// TIA Portal project "1905391_000_019" (V16)

(* hardware
DEVICE "S7-1200 station_1"  S7-1200 Station
   slot 0: "Rack_0"  S7-1200 Rack  Rack  V1.0
   slot 1: "PLC_1"  CPU 1211C DC/DC/DC  6ES7 211-1AE40-0XB0  V4.4
DEVICE "HMI_1"  TP900 Comfort
   slot 0: "HMI_1"  TP900 Comfort  6AV2 124-0JC01-0AX0  16.0.0.0
   slot 1: "HMI_RT_1"  TP900 Comfort  6AV2 124-0JC01-0AX0  16.0.0.0
   slot 5: "HMI_1.IE_CP_1"  PROFINET Interface  16.0.0.0
      slot 1: "PROFINET Interface_1"  PROFINET Interface
         slot 1: "Port_1"  Port
         slot 2: "Port_2"  Port
   slot 7: "HMI_1.MPI/DP_CP_1"  MPI/DP Interface  16.0.0.0
*)

// ===== PLC "PLC_1"  CPU 1211C DC/DC/DC =====

VAR_GLOBAL   // PLC tag table "Default tag table"
   "System_Byte" AT %MB1 : Byte;
   "FirstScan" AT %M1.0 : Bool;
   "DiagStatusUpdate" AT %M1.1 : Bool;
   "AlwaysTRUE" AT %M1.2 : Bool;
   "AlwaysFALSE" AT %M1.3 : Bool;
   "Clock_Byte" AT %MB0 : Byte;
   "Clock_10Hz" AT %M0.0 : Bool;
   "Clock_5Hz" AT %M0.1 : Bool;
   "Clock_2.5Hz" AT %M0.2 : Bool;
   "Clock_2Hz" AT %M0.3 : Bool;
   "Clock_1.25Hz" AT %M0.4 : Bool;
   "Clock_1Hz" AT %M0.5 : Bool;
   "Clock_0.625Hz" AT %M0.6 : Bool;
   "Clock_0.5Hz" AT %M0.7 : Bool;
END_VAR

VAR_GLOBAL CONSTANT   // PLC tag table "Default tag table"
   "STRING_LENGTH" : Int := 20;
   "ADP_PARAMETER_LENGTH" : Int := 5;
   "NULL_TOKEN" : Int := -1;
END_VAR

VAR_GLOBAL CONSTANT   // PLC tag table "Colors"
   "LABEL_COLOR" : String := '200_200_200';
   "DESELECTED_INPUT_COOR" : String := '250_250_250';
   "SELECTED_INPUT_COLOR" : String := '150,250,150';
   "BORDER_COLOR" : String := '200_200_200';
   "DIVIDER_COLOR" : String := '50_75_100';
   "THIS_SCREEN_COLOR" : String := '150;150;150';
   "OTHER_SCREEN_COLOR" : String := '100,100,100';
   "NAVIGATION_ACTUATE" : String := '150_250_150';
   "BACKGROUND_COLOR" : String := '150,150,200';
END_VAR

VAR_GLOBAL CONSTANT   // PLC tag table "Screen_Numbers"
   "WIRES_SCREEN_NUMBER" : Int := 1;
   "MATERIALS_SCREEN_NUMBER" : Int := 2;
END_VAR

TYPE "Divider.UDT"
   STRUCT
      background_animate : DInt;
      background_visible : Bool;
      line_animate : DInt;
      line_visible : Bool;
   END_STRUCT;
END_TYPE

TYPE "Row_Data.UDT"
   STRUCT
      background_animate : DInt;
      background_visible : Bool;
      cell_0_animate : DInt;
      cell_0_visible : Bool;
      cell_1_active : Bool;
      cell_1_animate : DInt;
      cell_1_enable : Bool;
      cell_1_input_finished : Bool;
      cell_1_value : String[50];
      cell_1_visible : Bool;
   END_STRUCT;
END_TYPE

TYPE "HMI_Interface.UDT"
   STRUCT
      materials : "Materials.HMI.UDT";
      meta : "HMI_Meta.UDT";
      navigation : "Navigation.HMI.UDT";
      wires : "Wire.HMI.UDT";
   END_STRUCT;
END_TYPE

TYPE "LED_Interface.UDT"
   STRUCT
      elements : "Material.LED.UDT";
      wires : "Wires.LED.UDT";
   END_STRUCT;
END_TYPE

TYPE "Navigation.HMI.UDT"
   STRUCT
      background_animate : DInt;
      background_visible : Bool;
      bottom_line_animate : DInt;
      bottom_line_visible : Bool;
      material_actuate : Bool;
      material_animate : DInt;
      material_cover_animate : DInt;
      material_cover_visible : Bool;
      material_enable : Bool;
      material_visible : Bool;
      wire_actuate : Bool;
      wire_animate : DInt;
      wire_cover_animate : DInt;
      wire_cover_visible : Bool;
      wire_enable : Bool;
      wire_visible : Bool;
   END_STRUCT;
END_TYPE

TYPE "Row_Custom.UDT"
   STRUCT
      background_animate : DInt;
      background_visible : Bool;
      cell_0_activate : Bool;
      cell_0_animate : DInt;
      cell_0_enable : Bool;
      cell_0_input_finished : Bool;
      cell_0_value : String[50];
      cell_0_visible : Bool;
      cell_1_activate : Bool;
      cell_1_animate : DInt;
      cell_1_enable : Bool;
      cell_1_input_finished : Bool;
      cell_1_value : String[50];
      cell_1_visible : Bool;
   END_STRUCT;
END_TYPE

TYPE "Row_Label.UDT"
   STRUCT
      background_animate : DInt;
      background_visible : Bool;
      cell_0_animate : DInt;
      cell_0_visible : Bool;
      cell_1_animate : DInt;
      cell_1_visible : Bool;
   END_STRUCT;
END_TYPE

TYPE "HMI_Meta.UDT"
   STRUCT
      screen_number : Int;
   END_STRUCT;
END_TYPE

TYPE "Screen_Background.UDT"
   STRUCT
      color : DInt;
      visible : Bool;
   END_STRUCT;
END_TYPE

// folder: ADP Data

TYPE "ADP.Row.2_Cells.UDT"
   STRUCT
      me : Array[0..1] of "ADP.Cell.UDT";
   END_STRUCT;
END_TYPE

TYPE "ADP.Cell.UDT"
   STRUCT
      color : String["ADP_PARAMETER_LENGTH"];
      flashing : String["ADP_PARAMETER_LENGTH"];
      h_align : String["ADP_PARAMETER_LENGTH"];
      lince_control : String["ADP_PARAMETER_LENGTH"];
      scroll_speed : String["ADP_PARAMETER_LENGTH"];
      size_and_face : String["ADP_PARAMETER_LENGTH"];
      v_align : String["ADP_PARAMETER_LENGTH"];
      value : String["STRING_LENGTH"];
   END_STRUCT;
END_TYPE

TYPE "ADP.Message_Buffer.UDT"
   STRUCT
      me : Array[0..999] of Byte;
   END_STRUCT;
END_TYPE

TYPE "ADP.Decoded.UDT"
   STRUCT
      color : "ADP.Decoded.Color.UDT";
      flash : "ADP.Decoded.Flash.UDT";
      horizontal_alignment : "ADP.Decoded.Horizontal_Alignment.UDT";
      line_control : "ADP.Decoded.Line_Control.UDT";
      scroll_speed : "ADP.Decoded.Scroll_Speed.UDT";
      size_and_face : "ADP.Decoded.Size_and_Face.UDT";
      vertical_alignment : "ADP.Decoded.Vertical_Alignment.UDT";
   END_STRUCT;
END_TYPE

TYPE "ADP.Decoded.Color.UDT"
   STRUCT
      black : String[8] := 'black';
      blue : String[8] := 'blue';
      green : String[8] := 'green';
      mix_1 : String[8] := 'mix 1';
      mix_2 : String[8] := 'mix 2';
      mix_3 : String[8] := 'mix 3';
      mix_4 : String[8] := 'mix 4';
      red : String[8] := 'red';
      white : String[8] := 'white';
      yellow : String[8] := 'yellow';
   END_STRUCT;
END_TYPE

TYPE "ADP.Decoded.Flash.UDT"
   STRUCT
      off : String[8] := 'off';
      on : String[8] := 'on';
   END_STRUCT;
END_TYPE

TYPE "ADP.Decoded.Horizontal_Alignment.UDT"
   STRUCT
      center : String[8] := 'center';
      left : String[8] := 'left';
      right : String[8] := 'right';
   END_STRUCT;
END_TYPE

TYPE "ADP.Encoded.UDT"
VERSION : 0.1
   STRUCT
      file_system : "ADP.Encoded.File_System.UDT";
      formatting : "ADP.Encoded.Formatting.UDT";
   END_STRUCT;
END_TYPE

TYPE "ADP.Message_Formats.Encoded.UDT"
   STRUCT
      color : String [5];
      flash : String [5];
      scroll_speed : String [5];
      size_and_face : String [5];
      vertical_alignment : String [5];
      horizontal_alignment : String [5];
   END_STRUCT;
END_TYPE

TYPE "ADP.Message_Formats.Decoded.UDT"
   STRUCT
      color : String [20];
      flash : String [20];
      scroll_speed : String [20];
      size_and_face : String [20];
      vertical_alignment : String [20];
      horizontal_alignment : String [20];
   END_STRUCT;
END_TYPE

TYPE "ADP.Decoded.Scroll_Speed.UDT"
   STRUCT
      slowest : String[9] := 'slowest';
      slow : String[9] := 'slow';
      normal : String[9] := 'normal';
      fast : String[9] := 'fast';
      fastest : String[9] := 'fastest';
   END_STRUCT;
END_TYPE

TYPE "ADP.Decoded.Size_and_Face.UDT"
   STRUCT
      bold_5 : String[11] := 'bold 5';
      bold_11 : String[11] := 'bold 11';
      bold_14 : String[11] := 'bold 14';
      bold_15 : String[11] := 'bold 15';
      bold_16 : String[11] := 'bold 16';
      bold_22 : String[11] := 'bold 22';
      bold_30 : String[11] := 'bold 30';
      bold_32 : String[11] := 'bold 32';
      bold_40 : String[11] := 'bold 40';
      normal_5 : String[11] := 'normal 5';
      normal_7 : String[11] := 'normal 7';
      normal_9 : String[11] := 'normal 9';
      normal_11 : String[11] := 'normal 11';
      normal_14 : String[11] := 'normal 14';
      normal_15 : String[11] := 'normal 15';
      normal_16 : String[11] := 'normal 16';
      normal_22 : String[11] := 'normal 22';
      normal_24 : String[11] := 'normal 24';
      normal_30 : String[11] := 'normal 30';
      normal_32 : String[11] := 'normal 32';
      normal_40 : String[11] := 'normal 40';
   END_STRUCT;
END_TYPE

TYPE "ADP.Decoded.Vertical_Alignment.UDT"
   STRUCT
      bottom_hold : String[15] := 'bottom hold';
      fill_hold : String[15] := 'fill hold';
      middle_hold : String[15] := 'middle hold';
      top_hold : String[15] := 'top hold';
      bottom_scroll : String[15] := 'bottom scroll';
      fill_scroll : String[15] := 'fill scroll';
      middle_scroll : String[15] := 'middle scroll';
      top_scroll : String[15] := 'top scroll';
   END_STRUCT;
END_TYPE

TYPE "ADP.Encoded.File_System.UDT"
   STRUCT
      "00 Start of Header" : String[5] := '$01';
      "01 Address" : String[5] := 'Z00';
      "02 Start of Text" : String[5] := '$02';
      "03 Command & File" : String[5] := 'AA';
      "04 END" : String[5] := '$04';
   END_STRUCT;
END_TYPE

TYPE "ADP.Encoded.Formatting.UDT"
   STRUCT
      color : "ADP.Encoded.Formatting.Color.UDT";
      flashing : "ADP.Encoded.Formatting.Flashing.UDT";
      horizontal_alignment : "ADP.Encoded.Formatting.Horizonta_Alignment.UDT";
      line_control : "ADP.Encoded.Formatting.Line_Control.UDT";
      scroll_speed : "ADP.Encoded.Formatting.Scroll_Speed.UDT";
      size_and_face : "ADP.Encoded.Formatting.Size_and_Face.UDT";
      vertical_alignment : "ADP.Encoded.Formatting.Vertical_Alignment.UDT";
   END_STRUCT;
END_TYPE

TYPE "ADP.Encoded.Formatting.Color.UDT"
   STRUCT
      black : String[5] := '$1C0';
      blue : String[5] := '$1C8';
      green : String[5] := '$1C2';
      mix_1 : String[5] := '$1C4';
      mix_2 : String[5] := '$1C5';
      mix_3 : String[5] := '$1C6';
      mix_4 : String[5] := '$1CY';
      red : String[5] := '$1C1';
      white : String[5] := '$1C9';
      yellow : String[5] := '$1C3';
   END_STRUCT;
END_TYPE

TYPE "ADP.Encoded.Formatting.Flashing.UDT"
   STRUCT
      off : String[5] := '$070';
      on : String[5] := '$071';
   END_STRUCT;
END_TYPE

TYPE "ADP.Encoded.Formatting.Size_and_Face.UDT"
   STRUCT
      bold_5 : String[5] := '$1AG';
      bold_11 : String[5] := '$1AH';
      bold_14 : String[5] := '$1A5';
      bold_15 : String[5] := '$1A6';
      bold_16 : String[5] := '$1A7';
      bold_22 : String[5] := '$1AC';
      bold_30 : String[5] := '$1AI';
      bold_32 : String[5] := '$1AJ';
      bold_40 : String[5] := '$1AK';
      normal_5 : String[5] := '$1A0';
      normal_7 : String[5] := '$1A1';
      normal_9 : String[5] := '$1A8';
      normal_11 : String[5] := '$1A9';
      normal_14 : String[5] := '$1A2';
      normal_15 : String[5] := '$1A3';
      normal_16 : String[5] := '$1A4';
      normal_22 : String[5] := '$1AA';
      normal_24 : String[5] := '$1AB';
      normal_30 : String[5] := '$1AD';
      normal_32 : String[5] := '$1AE';
      normal_40 : String[5] := '$1AF';
   END_STRUCT;
END_TYPE

TYPE "ADP.Encoded.Formatting.Horizonta_Alignment.UDT"
   STRUCT
      center : String[5] := '$L1';
      left : String[5] := '$L0';
      right : String[5] := '$L2';
   END_STRUCT;
END_TYPE

TYPE "ADP.Encoded.Formatting.Vertical_Alignment.UDT"
   STRUCT
      middle_hold : String[5] := '$1B b';
      fill_hold : String[5] := '$1B"b';
      bottom_hold : String[5] := '$1B&b';
      top_hold : String[5] := '$1B0b';
      bottom_scroll : String[5] := '$1B a';
      fill_scroll : String[5] := '$1B"a';
      middle_scroll : String[5] := '$1B&a';
      top_scroll : String[5] := '$1B0a';
   END_STRUCT;
END_TYPE

TYPE "ADP.Encoded.Formatting.Scroll_Speed.UDT"
   STRUCT
      slowest : String[5] := '$15';
      slow : String[5] := '$16';
      normal : String[5] := '$17';
      fast : String[5] := '$18';
      fastest : String[5] := '$19';
   END_STRUCT;
END_TYPE

TYPE "ADP.Encoded.Formatting.Line_Control.UDT"
   STRUCT
      new_line : String[5] := '$R';
      word_wrap : String[5] := '';
   END_STRUCT;
END_TYPE

TYPE "ADP.Decoded.Line_Control.UDT"
   STRUCT
      new_line : String[9] := 'new line';
      word_wrap : String[9] := 'word wrap';
   END_STRUCT;
END_TYPE

// folder: Material Data

TYPE "Materials.HMI.UDT"
   STRUCT
      background : "Screen_Background.UDT";
      bottom_border : "Divider.UDT";
      chromium : "Row_Data.UDT";
      custom : "Row_Custom.UDT";
      divider : "Divider.UDT";
      header : "Row_Label.UDT";
      heat : "Row_Data.UDT";
      manganese : "Row_Data.UDT";
      molybdenum : "Row_Data.UDT";
      nickel : "Row_Data.UDT";
      silicon : "Row_Data.UDT";
      vanadium : "Row_Data.UDT";
   END_STRUCT;
END_TYPE

TYPE "Material.Data.UDT"
   STRUCT
      chromium : Real;
      custom_value : Real;
      custom_name : String[50];
      heat : Real;
      manganese : Real;
      molybdenum : Real;
      nickel : Real;
      silicon : Real;
      vanadium : Real;
   END_STRUCT;
END_TYPE

TYPE "Material.LED.UDT"
   STRUCT
      chromium : "ADP.Row.2_Cells.UDT";
      custom : "ADP.Row.2_Cells.UDT";
      header : "ADP.Row.2_Cells.UDT";
      heat : "ADP.Row.2_Cells.UDT";
      manganese : "ADP.Row.2_Cells.UDT";
      molybdenum : "ADP.Row.2_Cells.UDT";
      nickel : "ADP.Row.2_Cells.UDT";
      silicon : "ADP.Row.2_Cells.UDT";
      vanadium : "ADP.Row.2_Cells.UDT";
   END_STRUCT;
   // chromium.me[0].value := 'chromium';
   // heat.me[0].value := 'heat';
   // manganese.me[0].value := 'manganese';
   // molybdenum.me[0].value := 'molybdenum';
   // nickel.me[0].value := 'nickel';
   // silicon.me[0].value := 'silicon';
   // vanadium.me[0].value := 'vanadium';
   // custom.me[0].value := 'Custom';
   // header.me[0].value := 'Material';
   // header.me[1].value := 'Bags';
END_TYPE

// folder: Wire Data

TYPE "Wire.UDT"
   STRUCT
      aluminum : Real;
      calcium_silicon : Real;
      carbon : Real;
      custom : Real;
      heat : Real;
      sulfur : Real;
   END_STRUCT;
END_TYPE

TYPE "Wires.LED.UDT"
   STRUCT
      aluminum : "ADP.Row.2_Cells.UDT";
      calcium_silicon : "ADP.Row.2_Cells.UDT";
      carbon : "ADP.Row.2_Cells.UDT";
      custom : "ADP.Row.2_Cells.UDT";
      heat : "ADP.Row.2_Cells.UDT";
      sulfur : "ADP.Row.2_Cells.UDT";
   END_STRUCT;
   // aluminum.me[0].value := 'AL Wire';
   // calcium_silicon.me[0].value := 'Cal/Sil Wire';
   // carbon.me[0].value := 'Carbon Wire';
   // heat.me[0].value := 'HEAT';
   // sulfur.me[0].value := 'Sulfur Wire';
   // custom.me[0].value := 'Custom';
END_TYPE

TYPE "Wire.HMI.UDT"
   STRUCT
      aluminum : "Row_Data.UDT";
      background : "Screen_Background.UDT";
      bottom_border : "Divider.UDT";
      calcium_silicon : "Row_Data.UDT";
      carbon : "Row_Data.UDT";
      divider : "Divider.UDT";
      header : "Row_Label.UDT";
      heat : "Row_Data.UDT";
      sulfur : "Row_Data.UDT";
   END_STRUCT;
END_TYPE

// folder: main/data

DATA_BLOCK "HMI_Interface.Data"   // DB2
{ S7_Optimized_Access := 'TRUE' }
VERSION : 0.1
BEGIN
   meta.screen_number := 1;
END_DATA_BLOCK

DATA_BLOCK "LED_Interface.Data"   // DB3
{ S7_Optimized_Access := 'TRUE' }
VERSION : 0.1
BEGIN
END_DATA_BLOCK

DATA_BLOCK "Display_IDB"   // DB4
{ S7_Optimized_Access := 'TRUE' }
VERSION : 0.1
// stored: InstanceOfName Display
"Display"
BEGIN
END_DATA_BLOCK

DATA_BLOCK "Middleware_IDB"   // DB5
{ S7_Optimized_Access := 'TRUE' }
VERSION : 0.1
// stored: InstanceOfName Middleware
"Middleware"
BEGIN
END_DATA_BLOCK

// folder: (top level)

ORGANIZATION_BLOCK "Main"   // OB1, LAD, ProgramCycle
TITLE = "Main Program Sweep (Cycle)"
{ S7_Optimized_Access := 'TRUE' }
VERSION : 0.1
   VAR_INPUT
      Initial_Call : Bool;   // Initial call of this OB
      Remanence : Bool;   // =True, if remanent data are available
   END_VAR
BEGIN

REGION Network 1
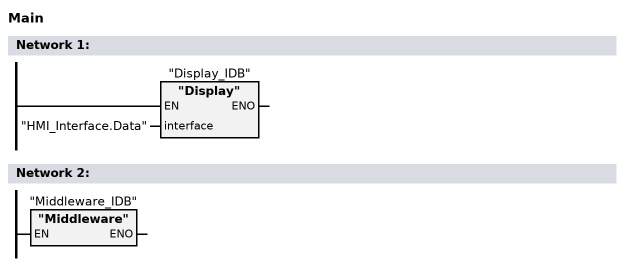
   RUNG wire#powerrail
      "Display_IDB"(interface := "HMI_Interface.Data")
   END_RUNG
   // the same network as SCL:
   "Display_IDB"(interface := "HMI_Interface.Data");   // "Display"
END_REGION

REGION Network 2
   RUNG wire#powerrail
      "Middleware_IDB"()
   END_RUNG
   // the same network as SCL:
   "Middleware_IDB"();   // "Middleware"
END_REGION
END_ORGANIZATION_BLOCK

ORGANIZATION_BLOCK "Startup"   // OB100, LAD, Startup
TITLE = "Complete Restart"
{ S7_Optimized_Access := 'TRUE' }
VERSION : 0.1
   VAR_INPUT
      LostRetentive : Bool;   // True if retentive data are lost
      LostRTC : Bool;   // True if date and time are lost
   END_VAR
BEGIN

REGION Network 1: INITIALIZE MATERIALS PAGE
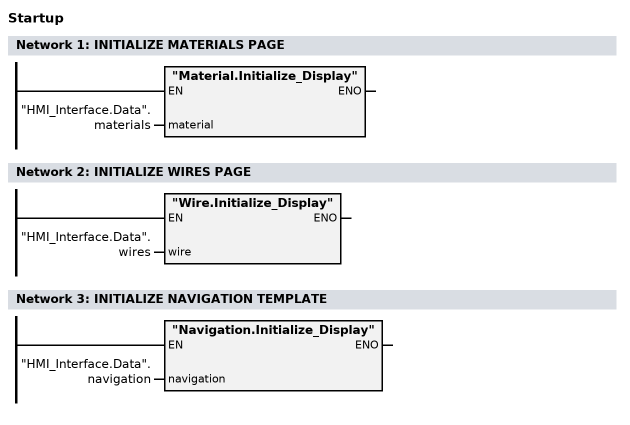
   RUNG wire#powerrail
      "Material.Initialize_Display"(material := "HMI_Interface.Data".materials)
   END_RUNG
   // the same network as SCL:
   "Material.Initialize_Display"(material := "HMI_Interface.Data".materials);
END_REGION

REGION Network 2: INITIALIZE WIRES PAGE
   RUNG wire#powerrail
      "Wire.Initialize_Display"(wire := "HMI_Interface.Data".wires)
   END_RUNG
   // the same network as SCL:
   "Wire.Initialize_Display"(wire := "HMI_Interface.Data".wires);
END_REGION

REGION Network 3: INITIALIZE NAVIGATION TEMPLATE
   RUNG wire#powerrail
      "Navigation.Initialize_Display"(navigation := "HMI_Interface.Data".navigation)
   END_RUNG
   // the same network as SCL:
   "Navigation.Initialize_Display"(navigation := "HMI_Interface.Data".navigation);
END_REGION
END_ORGANIZATION_BLOCK

// folder: any_data_types

FUNCTION "Any.Array.Length" : UDInt   // FC16, SCL
{ S7_Optimized_Access := 'TRUE' }
VERSION : 0.1
   VAR_INPUT
      "array" : Variant;
   END_VAR
   VAR_TEMP
      status : DInt;
      ret : UDInt;
   END_VAR
BEGIN
   #ret := CountOfElements(#array);
   #"Any.Array.Length" := #ret;
END_FUNCTION

// folder: bool

FUNCTION "Bool.Animate" : Void   // FC49, SCL
{ S7_Optimized_Access := 'TRUE' }
VERSION : 0.1
   VAR_INPUT
      signal : Bool;
      color_on : DInt;
      color_off : DInt;
   END_VAR
   VAR_IN_OUT
      animation : DInt;
   END_VAR
BEGIN
   IF #signal THEN
       #animation := #color_on;
       RETURN;
   END_IF;
   #animation := #color_off;
   RETURN;
END_FUNCTION

// folder: char

FUNCTION "Char.Is_Numeric" : Bool   // FC57, SCL
{ S7_Optimized_Access := 'TRUE' }
VERSION : 0.1
   VAR_INPUT
      character : Char;
   END_VAR
   VAR CONSTANT
      NUMBERS : String := '0123456789';
   END_VAR
BEGIN
   IF FIND(IN1 := #NUMBERS, IN2 := CHAR_TO_STRING(#character)) = 0 THEN
       #"Char.Is_Numeric" := FALSE;
       RETURN;
   END_IF;
   #"Char.Is_Numeric" := TRUE;
   RETURN;
END_FUNCTION

// folder: color

FUNCTION "Color.String_to_DInt" : DInt   // FC14, SCL
{ S7_Optimized_Access := 'TRUE' }
VERSION : 0.1
   VAR_INPUT
      color : String;   // enter rgb value with comma, semicolon, or underscore as delimeter. e.g.: '200,100,200' or '195_168_0'
   END_VAR
   VAR_TEMP
      _color : String;
      _background : DInt;
      _blue : DInt;
      _delimeters : Array[0..2] of String;
      _flash : DInt;
      _green : DInt;
      _red : DInt;
      _substrings : Array[0..3] of String;
   END_VAR
BEGIN
   REGION "COPY TO LOCAL"
       #_color := #color;
   END_REGION


   REGION "BACKGROUND MODE"
       #_background := 1;
       IF "Color.String_Is_Background"(#color) THEN
           #_background := -1;
           #_color := "String.Slice_Right"("string" := #_color,
                                           start_at := 1);
       END_IF;
   END_REGION


   REGION "SET UP DELIMETERS"
       #_delimeters[0] := ',';
       #_delimeters[1] := ';';
       #_delimeters[2] := '_';
   END_REGION


   REGION "SPLIT STRING"
       "String.Split_Multiple"(string_in := #_color,
                               delimeters := #_delimeters,
                               "pointer" := 0,
                               substrings => #_substrings);
       "String.Reverse_Array"(null_token := '',
                              string_array := #_substrings);
   END_REGION


   REGION "RETURN 0 ON INVALID STRING"
       IF NOT "Color.Validate_String"(#_substrings) THEN
           #"Color.String_to_DInt" := 0;
           RETURN;
       END_IF;
   END_REGION


   REGION "CALCULATE CODE"
       #_flash := STRING_TO_DINT(#_substrings[3]) * 1_000_000_000;
       #_red := STRING_TO_DINT(#_substrings[2]) * 1_000_000;
       #_green := STRING_TO_DINT(#_substrings[1]) * 1_000;
       #_blue := STRING_TO_DINT(#_substrings[0]);
   END_REGION


   REGION "RETURN"
       #"Color.String_to_DInt" := #_background * (#_flash + #_red + #_green + #_blue);
       RETURN;
   END_REGION
END_FUNCTION

FUNCTION "Color.Set_As_Background" : DInt   // FC27, SCL
{ S7_Optimized_Access := 'TRUE' }
VERSION : 0.1
   VAR_INPUT
      color_code : DInt;
   END_VAR
BEGIN
   IF #color_code < 0 THEN
       #"Color.Set_As_Background" := -1 * #color_code;
       RETURN;
   END_IF;
   #"Color.Set_As_Background" := #color_code;
   RETURN;
END_FUNCTION

FUNCTION "Color.Set_As_Foreground" : DInt   // FC30, SCL
{ S7_Optimized_Access := 'TRUE' }
VERSION : 0.1
   VAR_INPUT
      color_code : DInt;
   END_VAR
BEGIN
   IF #color_code >= 0 THEN
       #"Color.Set_As_Foreground" := -1 * #color_code;
       RETURN;
   END_IF;
   #"Color.Set_As_Foreground" := #color_code;
   RETURN;
END_FUNCTION

FUNCTION "Color.Flash_On" : DInt   // FC31, SCL
{ S7_Optimized_Access := 'TRUE' }
VERSION : 0.1
   VAR_INPUT
      color_code : DInt;
   END_VAR
   VAR CONSTANT
      FLASH : DInt := 1_000_000_000;
   END_VAR
BEGIN
   #"Color.Flash_On" := #FLASH + #color_code MOD #FLASH;
END_FUNCTION

FUNCTION "Color.Flash_Off" : DInt   // FC32, SCL
{ S7_Optimized_Access := 'TRUE' }
VERSION : 0.1
   VAR_INPUT
      color_code : DInt;
   END_VAR
   VAR CONSTANT
      FLASH : DInt := 1_000_000_000;
   END_VAR
BEGIN
   #"Color.Flash_Off" := #color_code MOD #FLASH;
END_FUNCTION

FUNCTION "Color.String_Is_Background" : Bool   // FC52, SCL
{ S7_Optimized_Access := 'TRUE' }
VERSION : 0.1
   VAR_INPUT
      color : String;
   END_VAR
BEGIN
   IF LEFT(IN := #color, L := 1) = '-' THEN
       #"Color.String_Is_Background" := TRUE;
       RETURN;
   END_IF;
   #"Color.String_Is_Background" := FALSE;
   RETURN;
END_FUNCTION

FUNCTION "Color.DInt_Is_Background" : Bool   // FC53, SCL
{ S7_Optimized_Access := 'TRUE' }
VERSION : 0.1
   VAR_INPUT
      color : DInt;
   END_VAR
BEGIN
   IF #color < 0 THEN
       #"Color.DInt_Is_Background" := FALSE;
       RETURN;
   END_IF;
   #"Color.DInt_Is_Background" := TRUE;
   RETURN;
END_FUNCTION

FUNCTION "Color.DInt_Is_Flashing" : Bool   // FC54, SCL
{ S7_Optimized_Access := 'TRUE' }
VERSION : 0.1
   VAR_INPUT
      color : DInt;
   END_VAR
   VAR CONSTANT
      FLASH : DInt := 1_000_000_000;
   END_VAR
BEGIN
   IF #color / #FLASH > 0 THEN
       #"Color.DInt_Is_Flashing" := TRUE;
       RETURN;
   END_IF;
   #"Color.DInt_Is_Flashing" := FALSE;
   RETURN;
END_FUNCTION

FUNCTION "Color.String_Is_Flashing" : Void   // FC55, SCL
{ S7_Optimized_Access := 'TRUE' }
VERSION : 0.1
   VAR_INPUT
      color : String;
   END_VAR
BEGIN
END_FUNCTION

FUNCTION "Color.Validate_String" : Bool   // FC56, SCL
{ S7_Optimized_Access := 'TRUE' }
VERSION : 0.1
   VAR_INPUT
      color : Array[*] of String;
   END_VAR
   VAR_TEMP
      _i : UDInt;
      _length : UDInt;
   END_VAR
BEGIN
   REGION "INVALID FLASH"
       IF #color[3] <> '1' AND #color[3] <> '' THEN
           #"Color.Validate_String" := FALSE;
           RETURN;
       END_IF;
   END_REGION


   REGION "NON-NUMERIC COMPONENT"
       FOR #_i := 0 TO #_length DO
           IF NOT "String.Is_Numeric"(#color[#_i]) THEN
               #"Color.Validate_String" := FALSE;
               RETURN;
           END_IF;
       END_FOR;
   END_REGION


   REGION "IS VALID"
       #"Color.Validate_String" := TRUE;
       RETURN;
   END_REGION
END_FUNCTION

// folder: divider

FUNCTION "Divider.Show" : Void   // FC2, SCL
{ S7_Optimized_Access := 'TRUE' }
VERSION : 0.1
   VAR_IN_OUT
      divider : "Divider.UDT";
   END_VAR
   VAR CONSTANT
      MODE : Bool := TRUE;
   END_VAR
BEGIN
   #divider.background_visible := #MODE;
   #divider.line_visible := #MODE;
END_FUNCTION

FUNCTION "Divider.Hide_Line" : Void   // FC13, SCL
{ S7_Optimized_Access := 'TRUE' }
VERSION : 0.1
   VAR_IN_OUT
      divider : "Divider.UDT";
   END_VAR
   VAR CONSTANT
      MODE : Bool := FALSE;
   END_VAR
BEGIN
   #divider.line_visible := #MODE;
END_FUNCTION

FUNCTION "Divider.Hide" : Void   // FC19, SCL
{ S7_Optimized_Access := 'TRUE' }
VERSION : 0.1
   VAR_IN_OUT
      divider : "Divider.UDT";
   END_VAR
   VAR CONSTANT
      MODE : Bool := FALSE;
   END_VAR
BEGIN
   #divider.background_visible := #MODE;
   #divider.line_visible := #MODE;
END_FUNCTION

FUNCTION "Divider.Initialize_Colors" : Void   // FC45, SCL
{ S7_Optimized_Access := 'TRUE' }
VERSION : 0.1
   VAR_IN_OUT
      divider : "Divider.UDT";
   END_VAR
BEGIN
   #divider.background_animate := "Color.String_to_DInt"("BORDER_COLOR");
   #divider.line_animate := "Color.String_to_DInt"("DIVIDER_COLOR");
END_FUNCTION

FUNCTION "Divider.Initialize" : Void   // FC46, SCL
{ S7_Optimized_Access := 'TRUE' }
VERSION : 0.1
   VAR_IN_OUT
      divider : "Divider.UDT";
   END_VAR
BEGIN
   "Divider.Show"(#divider);
   "Divider.Initialize_Colors"(#divider);
END_FUNCTION

// folder: main/display

FUNCTION_BLOCK "Display"   // FB5, SCL
{ S7_Optimized_Access := 'TRUE' }
VERSION : 0.1
   VAR_IN_OUT
      interface : "HMI_Interface.UDT";
   END_VAR
   VAR
      inst_HMI : "HMI";
   END_VAR
BEGIN
   REGION "HMI"
       #inst_HMI(interface := #interface);
   END_REGION

   REGION "LED"

   END_REGION
END_FUNCTION_BLOCK

// folder: main/display/HMI

FUNCTION_BLOCK "HMI"   // FB6, SCL
{ S7_Optimized_Access := 'TRUE' }
VERSION : 0.1
   VAR_IN_OUT
      interface : "HMI_Interface.UDT";
   END_VAR
   VAR
      place_holder : Bool;
   END_VAR
BEGIN
   REGION "VALIDATE INPUT"
       // not yet used
   END_REGION


   REGION "DISPLAY VALUES"
       // not yet used
   END_REGION


   REGION "ANIMATE"
       "HMI.Navigation"(interface := #interface);
       "HMI.Material"(#interface.materials);
       "HMI.Wire"(#interface.wires);
   END_REGION
END_FUNCTION_BLOCK

FUNCTION "HMI.Wire" : Void   // FC3, SCL
{ S7_Optimized_Access := 'TRUE' }
VERSION : 0.1
   VAR_IN_OUT
      wire : "Wire.HMI.UDT";
   END_VAR
BEGIN
   "Wire.Input_Animations"(#wire);
END_FUNCTION

FUNCTION "HMI.Material" : Void   // FC4, SCL
{ S7_Optimized_Access := 'TRUE' }
VERSION : 0.1
   VAR_IN_OUT
      material : "Materials.HMI.UDT";
   END_VAR
BEGIN
   "Material.Input_Animations"(#material);
END_FUNCTION

FUNCTION "HMI.Navigation" : Void   // FC8, SCL
{ S7_Optimized_Access := 'TRUE' }
VERSION : 0.1
   VAR_IN_OUT
      interface : "HMI_Interface.UDT";
   END_VAR
BEGIN
   "Navigation.Material_Acutation_Animation"(screen_number := #interface.meta.screen_number,
                                             navigation := #interface.navigation);
   "Navigation.Wire_Acutation_Animation"(screen_number := #interface.meta.screen_number,
                                         navigation := #interface.navigation);
   "Navigation.Wire_Cover_Animation"(screen_number := #interface.meta.screen_number,
                                     navigation := #interface.navigation);
END_FUNCTION

// folder: main/display/LED

FUNCTION_BLOCK "LED"   // FB7, SCL
{ S7_Optimized_Access := 'TRUE' }
VERSION : 0.1
   VAR
      Elements_Sign : "Elements_Sign";
      Wires_Sign : "Wires_Sign";
   END_VAR
BEGIN
   REGION "ELEMENTS"
       #Elements_Sign();
   END_REGION

   REGION "WIRES"
       #Wires_Sign();
   END_REGION
END_FUNCTION_BLOCK

FUNCTION_BLOCK "LED.Sign.Send"   // FB9, SCL
{ S7_Optimized_Access := 'TRUE' }
VERSION : 0.1
   VAR_INPUT
      data : "ADP.Message_Buffer.UDT";
      id : Conn_Ouc;
      request : Bool;
   END_VAR
   VAR
      TSEND : TSEND;
   END_VAR
BEGIN
   #TSEND(REQ := #request,
          ID := #id,
          DATA := #data);
END_FUNCTION_BLOCK

FUNCTION_BLOCK "LED.Sign"   // FB10, SCL
{ S7_Optimized_Access := 'TRUE' }
VERSION : 0.1
   VAR_INPUT
      id : Conn_Ouc;
      connection_parameters : TCON_Param;
      requests : Struct
         connect : Bool;
         diagnostics : Bool;
         disconnect : Bool;
         reset : Bool;
         send : Bool;
      END_STRUCT;
   END_VAR
   VAR
      Connect : "LED.Sign.Connect";
      Disconnect : "LED.Sign.Disconnect";
      Send : "LED.Sign.Send";
      Reset : "LED.Sign.Reset";
      Diagnostics : "LED.Sign.Diagnostics";
   END_VAR
BEGIN
   #Connect(request := #requests.connect,
            id := #id,
            connection_parameters := #connection_parameters);

   #Disconnect(id := #id,
               request := #requests.disconnect);

   #Send(id := #id,
         request := #requests.send);

   #Reset(id := #id,
          request := #requests.reset);

   #Diagnostics(id := #id,
                request := #requests.diagnostics);
END_FUNCTION_BLOCK

FUNCTION_BLOCK "LED.Sign.Connect"   // FB11, SCL
{ S7_Optimized_Access := 'TRUE' }
VERSION : 0.1
   VAR_INPUT
      request : Bool;
      id : Conn_Ouc;
      connection_parameters : TCON_Param;
   END_VAR
   VAR
      TCON : TCON;
   END_VAR
BEGIN
   #TCON(REQ := #request,
         ID := #id,
         CONNECT := #connection_parameters);
END_FUNCTION_BLOCK

FUNCTION_BLOCK "LED.Sign.Reset"   // FB12, SCL
{ S7_Optimized_Access := 'TRUE' }
VERSION : 0.1
   VAR_INPUT
      request : Bool;
      id : Conn_Ouc;
   END_VAR
   VAR
      T_RESET : T_RESET;
   END_VAR
BEGIN
   (* #T_RESET(REQ:=#request,
            ID:=#id,
            DONE=>_bool_out_,
            BUSY=>_bool_out_,
            ERROR=>_bool_out_,
            STATUS=>_word_out_); *)
END_FUNCTION_BLOCK

FUNCTION_BLOCK "LED.Sign.Disconnect"   // FB13, SCL
{ S7_Optimized_Access := 'TRUE' }
VERSION : 0.1
   VAR_INPUT
      request : Bool;
      id : Conn_Ouc;
   END_VAR
   VAR
      TDISCON : TDISCON;
   END_VAR
BEGIN
   #TDISCON(REQ := #request,
            ID := #id);
END_FUNCTION_BLOCK

FUNCTION_BLOCK "LED.Sign.Diagnostics"   // FB14, SCL
{ S7_Optimized_Access := 'TRUE' }
VERSION : 0.1
   VAR_INPUT
      request : Bool;
      id : Conn_Ouc;
   END_VAR
   VAR
      T_DIAG : T_DIAG;
   END_VAR
BEGIN
   #T_DIAG(REQ:=#request,
           ID:=#id);
END_FUNCTION_BLOCK

// folder: main/display/LED/Elements Sign

FUNCTION_BLOCK "Elements_Sign"   // FB16, SCL
{ S7_Optimized_Access := 'TRUE' }
VERSION : 0.1
   VAR
      Sign : "LED.Sign";
      id : Conn_Ouc;
      connection_parameters : TCON_Param;
   END_VAR
BEGIN
   "Elements_Sign.Assemble_Message"();
   #Sign(id := #id,
         connection_parameters := #connection_parameters);
END_FUNCTION_BLOCK

FUNCTION "Elements_Sign.Assemble_Message" : Void   // FC11, SCL
{ S7_Optimized_Access := 'TRUE' }
VERSION : 0.1
BEGIN
END_FUNCTION

// folder: main/display/LED/Wires Sign

FUNCTION_BLOCK "Wires_Sign"   // FB15, SCL
{ S7_Optimized_Access := 'TRUE' }
VERSION : 0.1
   VAR
      Sign : "LED.Sign";
      id : Conn_Ouc;
      connection_parameters : TCON_Param;
   END_VAR
BEGIN
   "Wires_Sign.Assemble_Message"();
   #Sign(id := #id,
         connection_parameters := #connection_parameters);
END_FUNCTION_BLOCK

FUNCTION "Wires_Sign.Assemble_Message" : Void   // FC12, SCL
{ S7_Optimized_Access := 'TRUE' }
VERSION : 0.1
BEGIN
END_FUNCTION

// folder: main/middleware

FUNCTION_BLOCK "Middleware"   // FB2, SCL
{ S7_Optimized_Access := 'TRUE' }
VERSION : 0.1
BEGIN
END_FUNCTION_BLOCK

// folder: material

FUNCTION "Material.Initialize_Display" : Void   // FC37, SCL
{ S7_Optimized_Access := 'TRUE' }
VERSION : 0.1
   VAR_IN_OUT
      material : "Materials.HMI.UDT";
   END_VAR
BEGIN
   "Screen_Background.Initialize"(#material.background);
   "Row_Data.Initialize"(#material.heat);
   "Row_Label.Initialize"(#material.header);
   "Divider.Initialize"(#material.divider);
   "Row_Data.Initialize"(#material.manganese);
   "Row_Data.Initialize"(#material.silicon);
   "Row_Data.Initialize"(#material.chromium);
   "Row_Data.Initialize"(#material.vanadium);
   "Row_Data.Initialize"(#material.nickel);
   "Row_Data.Initialize"(#material.molybdenum);
   "Row_Custom.Initialize"(#material.custom);
   "Divider.Initialize"(#material.bottom_border);
   "Divider.Hide_Line"(#material.bottom_border);
END_FUNCTION

FUNCTION "Material.Input_Animations" : Void   // FC76, SCL
{ S7_Optimized_Access := 'TRUE' }
VERSION : 0.1
   VAR_IN_OUT
      material : "Materials.HMI.UDT";
   END_VAR
BEGIN
   "Row_Data.Animate_In_Focus"(#material.heat);
   "Row_Data.Animate_In_Focus"(#material.manganese);
   "Row_Data.Animate_In_Focus"(#material.silicon);
   "Row_Data.Animate_In_Focus"(#material.chromium);
   "Row_Data.Animate_In_Focus"(#material.vanadium);
   "Row_Data.Animate_In_Focus"(#material.nickel);
   "Row_Data.Animate_In_Focus"(#material.molybdenum);
   "Row_Custom.Animate_In_Focus"(#material.custom);
END_FUNCTION

// folder: navigation

FUNCTION "Navigation.Initialize_Colors" : Void   // FC47, SCL
{ S7_Optimized_Access := 'TRUE' }
VERSION : 0.1
   VAR_IN_OUT
      navigation : "Navigation.HMI.UDT";
   END_VAR
BEGIN
   #navigation.background_animate := "Color.String_to_DInt"("BACKGROUND_COLOR");
   #navigation.bottom_line_animate := "Color.String_to_DInt"("DIVIDER_COLOR");
   #navigation.material_animate := "Color.String_to_DInt"("OTHER_SCREEN_COLOR");
   #navigation.material_cover_animate := "Color.String_to_DInt"("THIS_SCREEN_COLOR");
   #navigation.wire_animate := "Color.String_to_DInt"("THIS_SCREEN_COLOR");
   #navigation.wire_cover_animate := "Color.String_to_DInt"("THIS_SCREEN_COLOR");
END_FUNCTION

FUNCTION "Navigation.Wire_Acutation_Animation" : Void   // FC48, SCL
{ S7_Optimized_Access := 'TRUE' }
VERSION : 0.1
   VAR_INPUT
      screen_number : Int;
   END_VAR
   VAR_IN_OUT
      navigation : "Navigation.HMI.UDT";
   END_VAR
   VAR_TEMP
      _color_off : DInt;
   END_VAR
BEGIN
   CASE #screen_number OF
       "MATERIALS_SCREEN_NUMBER":
           #_color_off := "Color.String_to_DInt"("OTHER_SCREEN_COLOR");
       "WIRES_SCREEN_NUMBER":
           #_color_off := "Color.String_to_DInt"("THIS_SCREEN_COLOR");
   END_CASE;
   "Bool.Animate"(signal := #navigation.wire_actuate,
                  color_on := "Color.String_to_DInt"("NAVIGATION_ACTUATE"),
                  color_off := #_color_off,
                  animation := #navigation.wire_animate);
END_FUNCTION

FUNCTION "Navigation.Initialize_Visibility" : Void   // FC60, SCL
{ S7_Optimized_Access := 'TRUE' }
VERSION : 0.1
   VAR_IN_OUT
      navigation : "Navigation.HMI.UDT";
   END_VAR
BEGIN
   #navigation.background_visible := TRUE;
   #navigation.bottom_line_visible := TRUE;
   #navigation.material_visible := TRUE;
   #navigation.wire_visible := TRUE;
   #navigation.material_cover_visible := FALSE;
   #navigation.wire_cover_visible := TRUE;
END_FUNCTION

FUNCTION "Navigation.Initialize_Display" : Void   // FC61, SCL
{ S7_Optimized_Access := 'TRUE' }
VERSION : 0.1
   VAR_IN_OUT
      navigation : "Navigation.HMI.UDT";
   END_VAR
BEGIN
   "Navigation.Initialize_Colors"(#navigation);
   "Navigation.Initialize_Enable"(#navigation);
   "Navigation.Initialize_Visibility"(#navigation);
END_FUNCTION

FUNCTION "Navigation.Material_Acutation_Animation" : Void   // FC66, SCL
{ S7_Optimized_Access := 'TRUE' }
VERSION : 0.1
   VAR_INPUT
      screen_number : Int;
   END_VAR
   VAR_IN_OUT
      navigation : "Navigation.HMI.UDT";
   END_VAR
   VAR_TEMP
      _color_off : DInt;
   END_VAR
BEGIN
   CASE #screen_number OF
       "MATERIALS_SCREEN_NUMBER":
           #_color_off := "Color.String_to_DInt"("THIS_SCREEN_COLOR");
       "WIRES_SCREEN_NUMBER":
           #_color_off := "Color.String_to_DInt"("OTHER_SCREEN_COLOR");
   END_CASE;
   "Bool.Animate"(signal := #navigation.material_actuate,
                  color_on := "Color.String_to_DInt"("NAVIGATION_ACTUATE"),
                  color_off := #_color_off,
                  animation := #navigation.material_animate);
END_FUNCTION

FUNCTION "Navigation.Initialize_Enable" : Void   // FC69, SCL
{ S7_Optimized_Access := 'TRUE' }
VERSION : 0.1
   VAR_IN_OUT
      navigation : "Navigation.HMI.UDT";
   END_VAR
BEGIN
   #navigation.material_enable := TRUE;
   #navigation.wire_enable := TRUE;
END_FUNCTION

FUNCTION "Navigation.Wire_Cover_Animation" : Void   // FC73, SCL
{ S7_Optimized_Access := 'TRUE' }
VERSION : 0.1
   VAR_INPUT
      screen_number : Int;
   END_VAR
   VAR_IN_OUT
      navigation : "Navigation.HMI.UDT";
   END_VAR
BEGIN
   CASE #screen_number OF
       "MATERIALS_SCREEN_NUMBER":
           "Navigation.Bottom_Cover_Material_Screen"(#navigation);
       "WIRES_SCREEN_NUMBER":
           "Navigation.Bottom_Cover_Wire_Screen"(#navigation);
   END_CASE;
END_FUNCTION

FUNCTION "Navigation.Bottom_Cover_Wire_Screen" : Void   // FC74, SCL
{ S7_Optimized_Access := 'TRUE' }
VERSION : 0.1
   VAR_IN_OUT
      navigation : "Navigation.HMI.UDT";
   END_VAR
BEGIN
   #navigation.material_cover_visible := FALSE;
   #navigation.wire_cover_visible := TRUE;
END_FUNCTION

FUNCTION "Navigation.Bottom_Cover_Material_Screen" : Void   // FC75, SCL
{ S7_Optimized_Access := 'TRUE' }
VERSION : 0.1
   VAR_IN_OUT
      navigation : "Navigation.HMI.UDT";
   END_VAR
BEGIN
   #navigation.material_cover_visible := TRUE;
   #navigation.wire_cover_visible := FALSE;
END_FUNCTION

// folder: row_custom

FUNCTION "Row_Custom.Animate_In_Focus" : Void   // FC9, SCL
{ S7_Optimized_Access := 'TRUE' }
VERSION : 0.1
   VAR_IN_OUT
      row_custom : "Row_Custom.UDT";
   END_VAR
BEGIN
   "Bool.Animate"(signal := #row_custom.cell_0_activate,
                  color_on := "Color.String_to_DInt"("SELECTED_INPUT_COLOR"),
                  color_off := "Color.String_to_DInt"("DESELECTED_INPUT_COOR"),
                  animation := #row_custom.cell_0_animate);
   "Bool.Animate"(signal := #row_custom.cell_1_activate,
                  color_on := "Color.String_to_DInt"("SELECTED_INPUT_COLOR"),
                  color_off := "Color.String_to_DInt"("DESELECTED_INPUT_COOR"),
                  animation := #row_custom.cell_1_animate);
END_FUNCTION

FUNCTION "Row_Custom.Hide" : Void   // FC41, SCL
{ S7_Optimized_Access := 'TRUE' }
VERSION : 0.1
   VAR_IN_OUT
      row_custom : "Row_Custom.UDT";
   END_VAR
   VAR CONSTANT
      MODE : Bool := FALSE;
   END_VAR
BEGIN
   #row_custom.background_visible := #MODE;
   #row_custom.cell_0_visible := #MODE;
   #row_custom.cell_1_visible := #MODE;
END_FUNCTION

FUNCTION "Row_Custom.Enable" : Void   // FC42, SCL
{ S7_Optimized_Access := 'TRUE' }
VERSION : 0.1
   VAR_IN_OUT
      row_custom : "Row_Custom.UDT";
   END_VAR
   VAR CONSTANT
      MODE : Bool := TRUE;
   END_VAR
BEGIN
   #row_custom.cell_0_enable := #MODE;
   #row_custom.cell_1_enable := #MODE;
END_FUNCTION

FUNCTION "Row_Custom.Initialize_Colors" : Void   // FC43, SCL
{ S7_Optimized_Access := 'TRUE' }
VERSION : 0.1
   VAR_IN_OUT
      row_custom : "Row_Custom.UDT";
   END_VAR
BEGIN
   #row_custom.background_animate := "Color.String_to_DInt"("BORDER_COLOR");
   #row_custom.cell_0_animate := "Color.String_to_DInt"("DESELECTED_INPUT_COOR");
   #row_custom.cell_1_animate := "Color.String_to_DInt"("DESELECTED_INPUT_COOR");
END_FUNCTION

FUNCTION "Row_Custom.Initialize" : Void   // FC44, SCL
{ S7_Optimized_Access := 'TRUE' }
VERSION : 0.1
   VAR_IN_OUT
      row_custom : "Row_Custom.UDT";
   END_VAR
BEGIN
   "Row_Custom.Show"(#row_custom);
   "Row_Custom.Enable"(#row_custom);
   "Row_Custom.Initialize_Colors"(#row_custom);
END_FUNCTION

FUNCTION "Row_Custom.Show" : Void   // FC64, SCL
{ S7_Optimized_Access := 'TRUE' }
VERSION : 0.1
   VAR_IN_OUT
      row_custom : "Row_Custom.UDT";
   END_VAR
   VAR CONSTANT
      MODE : Bool := TRUE;
   END_VAR
BEGIN
   #row_custom.background_visible := #MODE;
   #row_custom.cell_0_visible := #MODE;
   #row_custom.cell_1_visible := #MODE;
END_FUNCTION

FUNCTION "Row_Custom.Disable" : Void   // FC65, SCL
{ S7_Optimized_Access := 'TRUE' }
VERSION : 0.1
   VAR_IN_OUT
      row_custom : "Row_Custom.UDT";
   END_VAR
   VAR CONSTANT
      MODE : Bool := FALSE;
   END_VAR
BEGIN
   #row_custom.cell_0_enable := #MODE;
   #row_custom.cell_1_enable := #MODE;
END_FUNCTION

FUNCTION "Row_Custom.Reset_Input_Finished" : Void   // FC78, SCL
{ S7_Optimized_Access := 'TRUE' }
VERSION : 0.1
   VAR_IN_OUT
      input_finished : Bool;
   END_VAR
BEGIN
   #input_finished := FALSE;
END_FUNCTION

// folder: row_data

FUNCTION "Row_Data.Initialize_Colors" : Void   // FC1, SCL
{ S7_Optimized_Access := 'TRUE' }
VERSION : 0.1
   VAR_IN_OUT
      row_data : "Row_Data.UDT";
   END_VAR
BEGIN
   #row_data.background_animate := "Color.String_to_DInt"("BORDER_COLOR");
   #row_data.cell_0_animate := "Color.String_to_DInt"("LABEL_COLOR");
   #row_data.cell_1_animate := "Color.String_to_DInt"("DESELECTED_INPUT_COOR");
END_FUNCTION

FUNCTION "Row_Data.Animate_In_Focus" : Void   // FC5, SCL
{ S7_Optimized_Access := 'TRUE' }
VERSION : 0.1
   VAR_IN_OUT
      row_data : "Row_Data.UDT";
   END_VAR
BEGIN
   "Bool.Animate"(signal := #row_data.cell_1_active,
                  color_on := "Color.String_to_DInt"("SELECTED_INPUT_COLOR"),
                  color_off := "Color.String_to_DInt"("DESELECTED_INPUT_COOR"),
                  animation := #row_data.cell_1_animate);
END_FUNCTION

FUNCTION "Row_Data.Show" : Void   // FC6, SCL
{ S7_Optimized_Access := 'TRUE' }
VERSION : 0.1
   VAR_IN_OUT
      row_data : "Row_Data.UDT";
   END_VAR
   VAR CONSTANT
      MODE : Bool := TRUE;
   END_VAR
BEGIN
   #row_data.background_visible := #MODE;
   #row_data.cell_0_visible := #MODE;
   #row_data.cell_1_visible := #MODE;
END_FUNCTION

FUNCTION "Row_Data.Enable" : Void   // FC7, SCL
{ S7_Optimized_Access := 'TRUE' }
VERSION : 0.1
   VAR_IN_OUT
      row_data : "Row_Data.UDT";
   END_VAR
   VAR CONSTANT
      MODE : Bool := TRUE;
   END_VAR
BEGIN
   #row_data.cell_1_enable := #MODE;
END_FUNCTION

FUNCTION "Row_Data.Hide" : Void   // FC23, SCL
{ S7_Optimized_Access := 'TRUE' }
VERSION : 0.1
   VAR_IN_OUT
      row_data : "Row_Data.UDT";
   END_VAR
   VAR CONSTANT
      MODE : Bool := FALSE;
   END_VAR
BEGIN
   #row_data.background_visible := #MODE;
   #row_data.cell_0_visible := #MODE;
   #row_data.cell_1_visible := #MODE;
END_FUNCTION

FUNCTION "Row_Data.Disable" : Void   // FC24, SCL
{ S7_Optimized_Access := 'TRUE' }
VERSION : 0.1
   VAR_IN_OUT
      row_data : "Row_Data.UDT";
   END_VAR
   VAR CONSTANT
      MODE : Bool := FALSE;
   END_VAR
BEGIN
   #row_data.cell_1_enable := #MODE;
END_FUNCTION

FUNCTION "Row_Data.Initialize" : Void   // FC28, SCL
{ S7_Optimized_Access := 'TRUE' }
VERSION : 0.1
   VAR_IN_OUT
      row_data : "Row_Data.UDT";
   END_VAR
BEGIN
   "Row_Data.Enable"(#row_data);
   "Row_Data.Initialize_Colors"(#row_data);
   "Row_Data.Show"(#row_data);
END_FUNCTION

FUNCTION "Row_Data.Reset_Input_Finished" : Void   // FC77, SCL
{ S7_Optimized_Access := 'TRUE' }
VERSION : 0.1
   VAR_IN_OUT
      row_data : "Row_Data.UDT";
   END_VAR
BEGIN
   #row_data.cell_1_input_finished := FALSE;
END_FUNCTION

// folder: row_label

FUNCTION "Row_Label.Show" : Void   // FC38, SCL
{ S7_Optimized_Access := 'TRUE' }
VERSION : 0.1
   VAR_IN_OUT
      row_label : "Row_Label.UDT";
   END_VAR
   VAR CONSTANT
      MODE : Bool := TRUE;
   END_VAR
BEGIN
   #row_label.background_visible := #MODE;
   #row_label.cell_0_visible := #MODE;
   #row_label.cell_1_visible := #MODE;
END_FUNCTION

FUNCTION "Row_Label.Initialize" : Void   // FC39, SCL
{ S7_Optimized_Access := 'TRUE' }
VERSION : 0.1
   VAR_IN_OUT
      row_label : "Row_Label.UDT";
   END_VAR
BEGIN
   "Row_Label.Show"(#row_label);
   "Row_Label.Initialize_Colors"(#row_label);
END_FUNCTION

FUNCTION "Row_Label.Initialize_Colors" : Void   // FC40, SCL
{ S7_Optimized_Access := 'TRUE' }
VERSION : 0.1
   VAR_IN_OUT
      row_label : "Row_Label.UDT";
   END_VAR
BEGIN
   #row_label.background_animate := "Color.String_to_DInt"("BORDER_COLOR");
   #row_label.cell_0_animate := "Color.String_to_DInt"("LABEL_COLOR");
   #row_label.cell_1_animate := "Color.String_to_DInt"("LABEL_COLOR");
END_FUNCTION

FUNCTION "Row_Label.Hide" : Void   // FC63, SCL
{ S7_Optimized_Access := 'TRUE' }
VERSION : 0.1
   VAR_IN_OUT
      row_label : "Row_Label.UDT";
   END_VAR
   VAR CONSTANT
      MODE : Bool := FALSE;
   END_VAR
BEGIN
   #row_label.background_visible := #MODE;
   #row_label.cell_0_visible := #MODE;
   #row_label.cell_1_visible := #MODE;
END_FUNCTION

// folder: screen_background

FUNCTION "Screen_Background.Initialize" : Void   // FC70, SCL
{ S7_Optimized_Access := 'TRUE' }
VERSION : 0.1
   VAR_IN_OUT
      background : "Screen_Background.UDT";
   END_VAR
BEGIN
   "Screen_Background.Initialize_Color"(#background);
   "Screen_Background.Initialize_Visibility"(#background);
END_FUNCTION

FUNCTION "Screen_Background.Initialize_Color" : Void   // FC71, SCL
{ S7_Optimized_Access := 'TRUE' }
VERSION : 0.1
   VAR_IN_OUT
      background : "Screen_Background.UDT";
   END_VAR
BEGIN
   #background.color := "Color.String_to_DInt"("THIS_SCREEN_COLOR");
END_FUNCTION

FUNCTION "Screen_Background.Initialize_Visibility" : Void   // FC72, SCL
{ S7_Optimized_Access := 'TRUE' }
VERSION : 0.1
   VAR_IN_OUT
      background : "Screen_Background.UDT";
   END_VAR
BEGIN
   #background.visible := TRUE;
END_FUNCTION

// folder: string

FUNCTION "String.Find" : Int   // FC18, SCL
{ S7_Optimized_Access := 'TRUE' }
VERSION : 0.1
   VAR_INPUT
      search_for : String;
      search_in : String;
   END_VAR
BEGIN
   #"String.Find" := FIND(IN1 := #search_in, IN2 := #search_for);
END_FUNCTION

FUNCTION "String.Strip_Sign" : String   // FC20, SCL
{ S7_Optimized_Access := 'TRUE' }
VERSION : 0.1
   VAR_INPUT
      "string" : String;
   END_VAR
   VAR_TEMP
      Length : Int;
      "String Box" : String;
      "Test Character" : String;
   END_VAR
   VAR CONSTANT
      "+" : Char := '+';
      "-" : Char := '-';
   END_VAR
BEGIN
   #"String Box" := #string;
   #"Test Character" := LEFT_STRING(IN := #"String Box",
                                    L := 1);
   IF #"Test Character" = #"+" OR #"Test Character" = #"-" THEN
       #Length := LEN(#"String Box");
       #"String Box" := RIGHT_STRING(IN := #"String Box", L := #Length - 1);

   END_IF;
   #"String.Strip_Sign" := #"String Box";
END_FUNCTION

FUNCTION "String.Trim" : String   // FC21, SCL
{ S7_Optimized_Access := 'TRUE' }
AUTHOR : Machado
FAMILY : String
VERSION : 1.0
// removes leading and trailing whitespace from input string
   VAR_INPUT
      "string" : String;
   END_VAR
   VAR_TEMP
      ret : String;
   END_VAR
   VAR CONSTANT
      space : String := ' ';
   END_VAR
BEGIN
   #ret := #string;
   WHILE LEFT(IN := #ret, L := 1) = #space DO
       #ret := RIGHT(IN := #ret, L := LEN(#ret) - 1);
   END_WHILE;
   WHILE RIGHT(IN := #ret, L := 1) = #space DO
       #ret := LEFT(IN := #ret, L := LEN(#ret) - 1);
   END_WHILE;
   #"String.Trim" := #ret;
END_FUNCTION

FUNCTION "String.Upper" : String   // FC22, SCL
{ S7_Optimized_Access := 'TRUE' }
AUTHOR : Machado
FAMILY : String
VERSION : 1.0
// returns the input string converted to all upper case
   VAR_INPUT
      "string" : String;
   END_VAR
   VAR_TEMP
      "type" : Bool;
      stringBox : String;
      status : Int;
      charArr : Array[0..255] of Char;
      cntChar : UInt;
      pChar : Int;
   END_VAR
   VAR CONSTANT
      asciiLow : Char := 'a';
      asciiHigh : Char := 'z';
      asciiCaseOffset : Int := 32;
   END_VAR
BEGIN
   Strg_TO_Chars(Strg := #string,
                 pChars := 0,
                 Cnt => #cntChar,
                 Chars := #charArr);

   FOR #pChar := 0 TO UINT_TO_INT(#cntChar) - 1 DO
       IF #asciiLow <= #charArr[#pChar] AND #charArr[#pChar] <= #asciiHigh THEN
           #charArr[#pChar] := INT_TO_CHAR(CHAR_TO_INT(#charArr[#pChar]) - #asciiCaseOffset);
       END_IF;
   END_FOR;

   Chars_TO_Strg(Chars := #charArr,
                 pChars := 0,
                 Cnt := #cntChar,
                 Strg => #stringBox);

   #"String.Upper" := #stringBox;
END_FUNCTION

FUNCTION "String.Split_Multiple" : Void   // FC26, SCL
{ S7_Optimized_Access := 'TRUE' }
VERSION : 0.1
   VAR_INPUT
      string_in : String;
      delimeters : Array[*] of String;
      pointer : Int;
   END_VAR
   VAR_OUTPUT
      substrings : Array[*] of String;
   END_VAR
   VAR_TEMP
      _i : Int;
      _position : Int;
      _return : String;
      _split : String;
   END_VAR
BEGIN
   REGION "GET POSITION OF DELIMETER IN STRING"
       #_position := "String.Find_Multiple.Breadth"(body := #string_in,
                                                    terms := #delimeters);
   END_REGION

   REGION "BASE CASE"
       IF #_position = 0 THEN
           #substrings[#pointer] := #string_in;
           "String.Split_Multiple.Clean_Output"("pointer" := #pointer + 1,
                                                substrings := #substrings);
           RETURN;
       END_IF;
   END_REGION


   REGION "RECURSIVE CASE"
       #substrings[#pointer] := LEFT(IN := #string_in, L := #_position);
       "String.Split_Multiple"(string_in := RIGHT(IN := #string_in, L := LEN(#string_in) - #_position),
                               delimeters := #delimeters,
                               "pointer" := #pointer + 1,
                               substrings => #substrings);
   END_REGION
END_FUNCTION

FUNCTION "String.Split_Single" : Void   // FC33, SCL
{ S7_Optimized_Access := 'TRUE' }
VERSION : 0.1
   VAR_INPUT
      string_in : String;
      delimeter : String;
      pointer : Int;
   END_VAR
   VAR_IN_OUT
      sub_strings : Array[*] of String;
   END_VAR
   VAR_TEMP
      _split : String;
      _position : Int;
      _return : String;
   END_VAR
BEGIN
   REGION "GET POSITION OF DELIMETER IN STRING"
       #_position := FIND(IN1 := #string_in,
                          IN2 := #delimeter);
   END_REGION

   REGION "BASE CASE"
       IF #_position = 0 THEN
           #sub_strings[#pointer] := #string_in;
           RETURN;
       END_IF;
   END_REGION


   REGION "RECURSIVE CASE"
       #sub_strings[#pointer] := LEFT(IN := #string_in, L := #_position - 1);
       "String.Split_Single"(string_in := RIGHT(IN := #string_in, L := LEN(#string_in) - #_position),
                             delimeter := #delimeter,
                             "pointer" := #pointer + 1,
                             sub_strings := #sub_strings);
   END_REGION
END_FUNCTION

FUNCTION "String.Find_Multiple.Breadth" : Int   // FC34, SCL
{ S7_Optimized_Access := 'TRUE' }
VERSION : 0.1
   VAR_INPUT
      body : String;
      terms : Array[*] of String;
   END_VAR
   VAR_TEMP
      _i : Int;
      _length : UDInt;
      _min : Int;
      _position : Int;
   END_VAR
   VAR CONSTANT
      BLANK : String;
   END_VAR
BEGIN
   (* 
       Depth first search of 'body' for first occurance of any element of 'terms'.
       For depth first search use WString.Find_Multiple.Depth.
       Returns character postion in the string (1 indexed).
       E.G.: 
           - body := WSTRING#'today?'
           - terms := <WSTRING#>['?', 'ay']
           - returns --> 6
       E.G.:
           - body := WSTRING#'today?'
           - terms := <WSTRING#>['ay', '?']
           - returns --> 4
   *)

   #_length := "Any.Array.Length"(#terms);

   IF #_length = 0 OR #body = #BLANK THEN
       #"String.Find_Multiple.Breadth" := 0;
       RETURN;
   END_IF;

   FOR #_i := 0 TO UDINT_TO_INT(#_length) - 1 DO
       #_position := FIND(IN1 := #body,
                          IN2 := #terms[#_i]);
       IF #_position = 0 THEN
           CONTINUE;
       END_IF;
       IF #_position < #_min OR #_min = 0 THEN
           #_min := #_position;
       END_IF;
   END_FOR;

   #"String.Find_Multiple.Breadth" := #_min;
END_FUNCTION

FUNCTION "String.Split_Multiple.Clean_Output" : Void   // FC35, SCL
{ S7_Optimized_Access := 'TRUE' }
VERSION : 0.1
   VAR_INPUT
      pointer : Int;
   END_VAR
   VAR_IN_OUT
      substrings : Array[*] of String;
   END_VAR
   VAR_TEMP
      _i : Int;
   END_VAR
   VAR CONSTANT
      BLANK : String;
   END_VAR
BEGIN
   FOR #_i := #"pointer" TO UDINT_TO_INT("Any.Array.Length"(#substrings)) - 1 DO
       #substrings[#_i] := #BLANK;
   END_FOR;
END_FUNCTION

FUNCTION "String.Search_Array" : Int   // FC50, SCL
{ S7_Optimized_Access := 'TRUE' }
VERSION : 0.1
   VAR_INPUT
      "array" : Array[*] of String;
      search_term : String;
   END_VAR
   VAR_TEMP
      _i : Int;
      _length : Int;
   END_VAR
BEGIN
   REGION "SEARCH ARRAY"    
       #_length := UDINT_TO_INT("Any.Array.Length"(#array)) - 1;
       FOR #_i := 0 TO #_length DO
           IF #array[#_i] = #search_term THEN
               #"String.Search_Array" := #_i;
               RETURN;
           END_IF;
       END_FOR;
   END_REGION

   REGION "RETURN"
       #"String.Search_Array" := "NULL_TOKEN";
       RETURN;
   END_REGION
END_FUNCTION

FUNCTION "String.Reverse_Array" : Void   // FC51, SCL
{ S7_Optimized_Access := 'TRUE' }
VERSION : 0.1
   VAR_INPUT
      null_token : String;
   END_VAR
   VAR_IN_OUT
      string_array : Array[*] of String;
   END_VAR
   VAR_TEMP
      _has_data_count : Int;
      _i : Int;
      _p_swap : Int;
      _temp : String;
   END_VAR
   VAR CONSTANT
      NOT_FOUND : Int := -1;
   END_VAR
BEGIN
   REGION "CHECK FOR FIRST EMPTY POSITION"
       #_has_data_count := "String.Search_Array"(array := #string_array,
                                                 search_term := #null_token);
   END_REGION


   REGION "EXIT ON EMPTY ARRAY"
       IF #_has_data_count = 0 THEN
           RETURN;
       END_IF;
   END_REGION


   REGION "ARRAY IS FULL"
       IF #_has_data_count = #NOT_FOUND THEN
           #_has_data_count := UDINT_TO_INT("Any.Array.Length"(#string_array));
       END_IF;
   END_REGION


   REGION "ADJUST TO ZERO INDEX"
       #_has_data_count -= 1;
   END_REGION


   REGION "SWAP ELEMENTS"
       FOR #_i := 0 TO #_has_data_count / 2 DO
           #_p_swap := #_has_data_count - #_i;
           #_temp := #string_array[#_i];
           #string_array[#_i] := #string_array[#_p_swap];
           #string_array[#_p_swap] := #_temp;
       END_FOR;
   END_REGION


   REGION "DONE"
       RETURN;
   END_REGION
END_FUNCTION

FUNCTION "String.Is_Numeric" : Bool   // FC58, SCL
{ S7_Optimized_Access := 'TRUE' }
VERSION : 0.1
   VAR_INPUT
      "string" : String;
   END_VAR
   VAR_TEMP
      _string : String;
   END_VAR
BEGIN
   #_string := #string;
   WHILE LEN(#_string) > 0 DO
       IF NOT "Char.Is_Numeric"(STRING_TO_CHAR(LEFT_STRING(IN := #_string, L := 1))) THEN
           #"String.Is_Numeric" := FALSE;
           RETURN;
       END_IF;
       #_string := "String.Slice_Right"("string" := #_string,
                                        start_at := 1);
   END_WHILE;
   #"String.Is_Numeric" := TRUE;
   RETURN;
END_FUNCTION

FUNCTION "String.Slice_Right" : String   // FC59, SCL
{ S7_Optimized_Access := 'TRUE' }
VERSION : 0.1
   VAR_INPUT
      "string" : String;
      start_at : Int;
   END_VAR
   VAR_TEMP
      _length : Int;
   END_VAR
BEGIN
   #"String.Slice_Right" := RIGHT_STRING(IN := #string,
                                         L := LEN(#string) - #start_at);
END_FUNCTION

FUNCTION "String.Count" : Int   // FC62, SCL
{ S7_Optimized_Access := 'TRUE' }
VERSION : 0.1
   VAR_INPUT
      space : String;   // count term ocuurances in space
      term : String;
   END_VAR
   VAR_TEMP
      _count : Int;
      _position : Int;
      _space : String;
   END_VAR
BEGIN
   #_space := #space;
   #_position := FIND(IN1 := #_space,
                      IN2 := #term);
   IF #_position = 0 THEN
       #"String.Count" := 0;
       RETURN;
   END_IF;
   WHILE #_position > 0 DO
       #_count += 1;
       #_space := RIGHT(IN := #_space,
                        L := LEN(#_space) - #_position);
       #_position := FIND(IN1 := #_space,
                          IN2 := #term);
   END_WHILE;
   #"String.Count" := #_count;
   RETURN;
END_FUNCTION

// folder: wire

FUNCTION "Wire.Input_Animations" : Void   // FC10, SCL
{ S7_Optimized_Access := 'TRUE' }
VERSION : 0.1
   VAR_IN_OUT
      wire : "Wire.HMI.UDT";
   END_VAR
BEGIN
   "Row_Data.Animate_In_Focus"(#wire.heat);
   "Row_Data.Animate_In_Focus"(#wire.carbon);
   "Row_Data.Animate_In_Focus"(#wire.calcium_silicon);
   "Row_Data.Animate_In_Focus"(#wire.aluminum);
   "Row_Data.Animate_In_Focus"(#wire.sulfur);
END_FUNCTION

FUNCTION "Wire.Initialize_Display" : Void   // FC29, SCL
{ S7_Optimized_Access := 'TRUE' }
VERSION : 0.1
   VAR_IN_OUT
      wire : "Wire.HMI.UDT";
   END_VAR
BEGIN
   "Screen_Background.Initialize"(#wire.background);
   "Row_Data.Initialize"(#wire.heat);
   "Row_Label.Initialize"(#wire.header);
   "Divider.Initialize"(#wire.divider);
   "Row_Data.Initialize"(#wire.carbon);
   "Row_Data.Initialize"(#wire.calcium_silicon);
   "Row_Data.Initialize"(#wire.aluminum);
   "Row_Data.Initialize"(#wire.sulfur);
   "Divider.Initialize"(#wire.bottom_border);
   "Divider.Hide_Line"(#wire.bottom_border);
END_FUNCTION

// folder: wstring

FUNCTION "WString.Split_Single" : Void   // FC15, SCL
{ S7_Optimized_Access := 'TRUE' }
VERSION : 0.1
   VAR_INPUT
      wstring_in : WString;
      delimeter : WString;
      pointer : Int;
   END_VAR
   VAR_IN_OUT
      sub_strings : Array[*] of WString;
   END_VAR
   VAR_TEMP
      _split : WString;
      _position : Int;
      _return : WString;
   END_VAR
BEGIN
   REGION "GET POSITION OF DELIMETER IN STRING"
       #_position := FIND(IN1 := #wstring_in,
                          IN2 := #delimeter);
   END_REGION

   REGION "BASE CASE"
       IF #_position = 0 THEN
           #sub_strings[#pointer] := #wstring_in;
           RETURN;
       END_IF;
   END_REGION


   REGION "RECURSIVE CASE"
       #sub_strings[#pointer] := LEFT(IN := #wstring_in, L := #_position - 1);
       "WString.Split_Single"(wstring_in := RIGHT(IN := #wstring_in, L := LEN(#wstring_in) - #_position),
                              delimeter := #delimeter,
                              "pointer" := #pointer + 1,
                              sub_strings := #sub_strings);
   END_REGION
END_FUNCTION

FUNCTION "WString.Find_Multiple.Breadth" : Int   // FC17, SCL
{ S7_Optimized_Access := 'TRUE' }
VERSION : 0.1
   VAR_INPUT
      body : WString;
      terms : Array[*] of WString[1];
   END_VAR
   VAR_TEMP
      _i : Int;
      _length : UDInt;
      _min : Int;
      _position : Int;
   END_VAR
   VAR CONSTANT
      BLANK : WString;
   END_VAR
BEGIN
   (* 
       Depth first search of 'body' for first occurance of any element of 'terms'.
       For depth first search use WString.Find_Multiple.Depth.
       Returns character postion in the string (1 indexed).
       E.G.: 
           - body := WSTRING#'today?'
           - terms := <WSTRING#>['?', 'ay']
           - returns --> 6
       E.G.:
           - body := WSTRING#'today?'
           - terms := <WSTRING#>['ay', '?']
           - returns --> 4
   *)

   #_length := "Any.Array.Length"(#terms);

   IF #_length = 0 OR #body = #BLANK THEN
       #"WString.Find_Multiple.Breadth" := 0;
       RETURN;
   END_IF;

   FOR #_i := 0 TO UDINT_TO_INT(#_length) - 1 DO
       #_position := FIND(IN1 := #body,
                          IN2 := #terms[#_i]);
       IF #_position = 0 THEN
           CONTINUE;
       END_IF;
       IF #_position < #_min OR #_min = 0 THEN
           #_min := #_position;
       END_IF;
   END_FOR;

   #"WString.Find_Multiple.Breadth" := #_min;
END_FUNCTION

FUNCTION "WString.Split_Multiple.Clean_Output" : Void   // FC25, SCL
{ S7_Optimized_Access := 'TRUE' }
VERSION : 0.1
   VAR_INPUT
      pointer : Int;
   END_VAR
   VAR_IN_OUT
      substrings : Array[*] of WString[20];
   END_VAR
   VAR_TEMP
      _i : Int;
   END_VAR
   VAR CONSTANT
      BLANK : WString;
   END_VAR
BEGIN
   FOR #_i := #"pointer" TO UDINT_TO_INT("Any.Array.Length"(#substrings)) - 1 DO
       #substrings[#_i] := wstring#'';
   END_FOR;
END_FUNCTION

FUNCTION "WString.Split_Multiple" : Void   // FC36, SCL
{ S7_Optimized_Access := 'TRUE' }
VERSION : 0.1
   VAR_INPUT
      wstring_in : WString;
      delimeters : Array[*] of WString[1];
      pointer : Int;
   END_VAR
   VAR_OUTPUT
      substrings : Array[*] of WString[20];
   END_VAR
   VAR_TEMP
      _i : Int;
      _position : Int;
      _return : WString;
      _split : WString;
   END_VAR
BEGIN
   REGION "GET POSITION OF DELIMETER IN STRING"
       #_position := "WString.Find_Multiple.Breadth"(body := #wstring_in,
                                                     terms := #delimeters);
   END_REGION

   REGION "BASE CASE"
       IF #_position = 0 THEN
           #substrings[#pointer] := #wstring_in;
           "WString.Split_Multiple.Clean_Output"("pointer" := #pointer + 1,
                                                 substrings := #substrings);
           RETURN;
       END_IF;
   END_REGION


   REGION "RECURSIVE CASE"
       #substrings[#pointer] := LEFT(IN := #wstring_in, L := #_position);
       "WString.Split_Multiple"(wstring_in := RIGHT(IN := #wstring_in, L := LEN(#wstring_in) - #_position),
                                delimeters := #delimeters,
                                "pointer" := #pointer + 1,
                                substrings => #substrings);
   END_REGION
END_FUNCTION

FUNCTION "WString.Search_Array" : Int   // FC67, SCL
{ S7_Optimized_Access := 'TRUE' }
VERSION : 0.1
   VAR_INPUT
      "array" : Array[*] of WString;
      search_term : WString;
   END_VAR
   VAR_TEMP
      _i : Int;
      _length : Int;
   END_VAR
BEGIN
   REGION "SEARCH ARRAY"    
       #_length := UDINT_TO_INT("Any.Array.Length"(#array)) - 1;
       FOR #_i := 0 TO #_length DO
           IF #array[#_i] = #search_term THEN
               #"WString.Search_Array" := #_i;
               RETURN;
           END_IF;
       END_FOR;
   END_REGION

   REGION "RETURN"
       #"WString.Search_Array" := "NULL_TOKEN";
       RETURN;
   END_REGION
END_FUNCTION

FUNCTION "WString.Reverse_Array" : Void   // FC68, SCL
{ S7_Optimized_Access := 'TRUE' }
VERSION : 0.1
   VAR_INPUT
      null_token : WString;
   END_VAR
   VAR_IN_OUT
      wstring_array : Array[*] of WString;
   END_VAR
   VAR_TEMP
      _has_data_count : Int;
      _i : Int;
      _p_swap : Int;
      _temp : WString;
   END_VAR
   VAR CONSTANT
      NOT_FOUND : Int := -1;
   END_VAR
BEGIN
   REGION "CHECK FOR FIRST EMPTY POSITION"
       #_has_data_count := "WString.Search_Array"(array := #wstring_array,
                                                  search_term := #null_token);
   END_REGION


   REGION "EXIT ON EMPTY ARRAY"
       IF #_has_data_count = 0 THEN
           RETURN;
       END_IF;
   END_REGION


   REGION "ARRAY IS FULL"
       IF #_has_data_count = #NOT_FOUND THEN
           #_has_data_count := UDINT_TO_INT("Any.Array.Length"(#wstring_array));
       END_IF;
   END_REGION


   REGION "ADJUST TO ZERO INDEX"
       #_has_data_count -= 1;
   END_REGION


   REGION "SWAP ELEMENTS"
       FOR #_i := 0 TO #_has_data_count / 2 DO
           #_p_swap := #_has_data_count - #_i;
           #_temp := #wstring_array[#_i];
           #wstring_array[#_i] := #wstring_array[#_p_swap];
           #wstring_array[#_p_swap] := #_temp;
       END_FOR;
   END_REGION


   REGION "DONE"
       RETURN;
   END_REGION
END_FUNCTION

// ===== library types =====

TYPE "Row.UDT"
   STRUCT
      background_animate : DInt;
      background_visible : Bool;
      cell_0_animate : DInt;
      cell_0_visible : Bool;
      cell_1_active : Bool;
      cell_1_animate : DInt;
      cell_1_enable : Bool;
      cell_1_input_finished : Bool;
      cell_1_value : String[50];
      cell_1_visible : Bool;
   END_STRUCT;
END_TYPE

TYPE "Navigation.UDT"
   STRUCT
      background_animate : DInt;
      background_visible : Bool;
      bottom_line_animate : DInt;
      bottom_line_visible : Bool;
      material_actuate : Bool;
      material_animate : DInt;
      material_cover_animate : DInt;
      material_cover_visible : Bool;
      material_enable : Bool;
      material_visible : Bool;
      wire_actuate : Bool;
      wire_animate : DInt;
      wire_cover_animate : DInt;
      wire_cover_visible : Bool;
      wire_enable : Bool;
      wire_visible : Bool;
   END_STRUCT;
END_TYPE

FUNCTION "Array.Any.Length" : UDInt   // FC16, SCL
{ S7_Optimized_Access := 'TRUE' }
VERSION : 0.1
   VAR_INPUT
      "array" : Variant;
   END_VAR
   VAR_TEMP
      status : DInt;
      ret : UDInt;
   END_VAR
BEGIN
   #ret := CountOfElements(#array);
   #"Array.Any.Length" := #ret;
END_FUNCTION

// folder: color

FUNCTION "Color.Decode_String" : DInt   // FC14, SCL
{ S7_Optimized_Access := 'TRUE' }
VERSION : 0.1
   VAR_INPUT
      color : String;   // enter rgb value with comma, semicolon, or underscore as delimeter. e.g.: '200,100,200' or '195_168_0'
   END_VAR
   VAR_TEMP
      _delimeters : Array[0..2] of String[1];
      _substrings : Array[0..2] of String[20];
      _red : DInt;
      _green : DInt;
      _blue : DInt;
   END_VAR
BEGIN
   #_delimeters[0] := ',';
   #_delimeters[1] := ';';
   #_delimeters[2] := '_';
   "String.Split_Multiple"(string_in:=#color,
                           delimeters:=#_delimeters,
                           "pointer":=0,
                           substrings=>#_substrings);
   #_red := STRING_TO_DINT(#_substrings[0]) * 1_000_000;
   #_green := STRING_TO_DINT(#_substrings[1]) * 1_000;
   #_blue := STRING_TO_DINT(#_substrings[2]);
   #"Color.Decode_String" := #_red + #_green + #_blue;
END_FUNCTION

// ===== library: MasterCopy "Copy of PLC data types in ADP Data" =====

// folder: ADP Data

TYPE "ADP: Encoded"
VERSION : 0.1
   STRUCT
      file_system : "ADP: Encoded: File System";
      formatting : "ADP: Encoded: Formatting";
   END_STRUCT;
END_TYPE

TYPE "ADP: Decoded"
   STRUCT
      color : "ADP: Decoded: Color";
      flash : "ADP: Decoded: Flash";
      horizontal_alignment : "ADP: Decoded: Horizontal Alignment";
      line_control : "ADP: Decoded: Line Control";
      scroll_speed : "ADP: Decoded: Scroll Speed";
      size_and_face : "ADP: Decoded: Size and Face";
      vertical_alignment : "ADP: Decoded: Vertical Alignment";
   END_STRUCT;
END_TYPE

TYPE "ADP: Decoded: Color"
   STRUCT
      black : String[8] := 'black';
      blue : String[8] := 'blue';
      green : String[8] := 'green';
      mix_1 : String[8] := 'mix 1';
      mix_2 : String[8] := 'mix 2';
      mix_3 : String[8] := 'mix 3';
      mix_4 : String[8] := 'mix 4';
      red : String[8] := 'red';
      white : String[8] := 'white';
      yellow : String[8] := 'yellow';
   END_STRUCT;
END_TYPE

TYPE "ADP: Decoded: Flash"
   STRUCT
      off : String[8] := 'off';
      on : String[8] := 'on';
   END_STRUCT;
END_TYPE

TYPE "ADP: Decoded: Horizontal Alignment"
   STRUCT
      center : String[8] := 'center';
      left : String[8] := 'left';
      right : String[8] := 'right';
   END_STRUCT;
END_TYPE

TYPE "ADP: Message Formats: Encoded"
   STRUCT
      color : String [5];
      flash : String [5];
      scroll_speed : String [5];
      size_and_face : String [5];
      vertical_alignment : String [5];
      horizontal_alignment : String [5];
   END_STRUCT;
END_TYPE

TYPE "ADP: Message Formats: Decoded"
   STRUCT
      color : String [20];
      flash : String [20];
      scroll_speed : String [20];
      size_and_face : String [20];
      vertical_alignment : String [20];
      horizontal_alignment : String [20];
   END_STRUCT;
END_TYPE

TYPE "ADP: Decoded: Scroll Speed"
   STRUCT
      slowest : String[9] := 'slowest';
      slow : String[9] := 'slow';
      normal : String[9] := 'normal';
      fast : String[9] := 'fast';
      fastest : String[9] := 'fastest';
   END_STRUCT;
END_TYPE

TYPE "ADP: Decoded: Size and Face"
   STRUCT
      bold_5 : String[11] := 'bold 5';
      bold_11 : String[11] := 'bold 11';
      bold_14 : String[11] := 'bold 14';
      bold_15 : String[11] := 'bold 15';
      bold_16 : String[11] := 'bold 16';
      bold_22 : String[11] := 'bold 22';
      bold_30 : String[11] := 'bold 30';
      bold_32 : String[11] := 'bold 32';
      bold_40 : String[11] := 'bold 40';
      normal_5 : String[11] := 'normal 5';
      normal_7 : String[11] := 'normal 7';
      normal_9 : String[11] := 'normal 9';
      normal_11 : String[11] := 'normal 11';
      normal_14 : String[11] := 'normal 14';
      normal_15 : String[11] := 'normal 15';
      normal_16 : String[11] := 'normal 16';
      normal_22 : String[11] := 'normal 22';
      normal_24 : String[11] := 'normal 24';
      normal_30 : String[11] := 'normal 30';
      normal_32 : String[11] := 'normal 32';
      normal_40 : String[11] := 'normal 40';
   END_STRUCT;
END_TYPE

TYPE "ADP: Decoded: Vertical Alignment"
   STRUCT
      bottom_hold : String[15] := 'bottom hold';
      fill_hold : String[15] := 'fill hold';
      middle_hold : String[15] := 'middle hold';
      top_hold : String[15] := 'top hold';
      bottom_scroll : String[15] := 'bottom scroll';
      fill_scroll : String[15] := 'fill scroll';
      middle_scroll : String[15] := 'middle scroll';
      top_scroll : String[15] := 'top scroll';
   END_STRUCT;
END_TYPE

TYPE "ADP: Encoded: File System"
   STRUCT
      "00 Start of Header" : String[5] := '$01';
      "01 Address" : String[5] := 'Z00';
      "02 Start of Text" : String[5] := '$02';
      "03 Command & File" : String[5] := 'AA';
      "04 END" : String[5] := '$04';
   END_STRUCT;
END_TYPE

TYPE "ADP: Encoded: Formatting"
   STRUCT
      color : "ADP: Encoded: Formatting: Color";
      flashing : "ADP: Encoded: Formatting: Flashing";
      horizontal_alignment : "ADP: Encoded: Formatting: Horizontal Alignment";
      line_control : "ADP: Encoded: Formatting: Line Control";
      scroll_speed : "ADP: Encoded: Formatting: Scroll Speed";
      size_and_face : "ADP: Encoded: Formatting: Size and Face";
      vertical_alignment : "ADP: Encoded: Formatting: Vertical Alignment";
   END_STRUCT;
END_TYPE

TYPE "ADP: Encoded: Formatting: Color"
   STRUCT
      black : String[5] := '$1C0';
      blue : String[5] := '$1C8';
      green : String[5] := '$1C2';
      mix_1 : String[5] := '$1C4';
      mix_2 : String[5] := '$1C5';
      mix_3 : String[5] := '$1C6';
      mix_4 : String[5] := '$1CY';
      red : String[5] := '$1C1';
      white : String[5] := '$1C9';
      yellow : String[5] := '$1C3';
   END_STRUCT;
END_TYPE

TYPE "ADP: Encoded: Formatting: Flashing"
   STRUCT
      off : String[5] := '$070';
      on : String[5] := '$071';
   END_STRUCT;
END_TYPE

TYPE "ADP: Encoded: Formatting: Size and Face"
   STRUCT
      bold_5 : String[5] := '$1AG';
      bold_11 : String[5] := '$1AH';
      bold_14 : String[5] := '$1A5';
      bold_15 : String[5] := '$1A6';
      bold_16 : String[5] := '$1A7';
      bold_22 : String[5] := '$1AC';
      bold_30 : String[5] := '$1AI';
      bold_32 : String[5] := '$1AJ';
      bold_40 : String[5] := '$1AK';
      normal_5 : String[5] := '$1A0';
      normal_7 : String[5] := '$1A1';
      normal_9 : String[5] := '$1A8';
      normal_11 : String[5] := '$1A9';
      normal_14 : String[5] := '$1A2';
      normal_15 : String[5] := '$1A3';
      normal_16 : String[5] := '$1A4';
      normal_22 : String[5] := '$1AA';
      normal_24 : String[5] := '$1AB';
      normal_30 : String[5] := '$1AD';
      normal_32 : String[5] := '$1AE';
      normal_40 : String[5] := '$1AF';
   END_STRUCT;
END_TYPE

TYPE "ADP: Encoded: Formatting: Horizontal Alignment"
   STRUCT
      center : String[5] := '$L1';
      left : String[5] := '$L0';
      right : String[5] := '$L2';
   END_STRUCT;
END_TYPE

TYPE "ADP: Encoded: Formatting: Vertical Alignment"
   STRUCT
      middle_hold : String[5] := '$1B b';
      fill_hold : String[5] := '$1B"b';
      bottom_hold : String[5] := '$1B&b';
      top_hold : String[5] := '$1B0b';
      bottom_scroll : String[5] := '$1B a';
      fill_scroll : String[5] := '$1B"a';
      middle_scroll : String[5] := '$1B&a';
      top_scroll : String[5] := '$1B0a';
   END_STRUCT;
END_TYPE

TYPE "ADP: Encoded: Formatting: Scroll Speed"
   STRUCT
      slowest : String[5] := '$15';
      slow : String[5] := '$16';
      normal : String[5] := '$17';
      fast : String[5] := '$18';
      fastest : String[5] := '$19';
   END_STRUCT;
END_TYPE

TYPE "ADP: Encoded: Formatting: Line Control"
   STRUCT
      new_line : String[5] := '$R';
      word_wrap : String[5] := '';
   END_STRUCT;
END_TYPE

TYPE "ADP: Decoded: Line Control"
   STRUCT
      new_line : String[9] := 'new line';
      word_wrap : String[9] := 'word wrap';
   END_STRUCT;
END_TYPE

(* ===== HMI "HMI_RT_1" =====
system functions are stored by id; their names below are inferred from use
connection "HMI_Connection_1": ETHERNET, S7_1200_OMS

HMI tags "Default tag table"
   "Clock_Byte" : Byte = PLC Clock_Byte AT %MB0, 100 ms
   "HMI_Interface.Data_materials" : Materials.HMI.UDT = PLC "HMI_Interface.Data".materials AT %DB1.DBB0, 100 ms
   "HMI_Interface.Data_navigation" : Navigation.HMI.UDT = PLC "HMI_Interface.Data".navigation AT %DB1.DBW0, 100 ms
   "HMI_Interface.Data_wires" : Wire.HMI.UDT = PLC "HMI_Interface.Data".wires AT %DB1.DBW0, 100 ms
   "HMI_Interface.Data_meta" : HMI_Meta.UDT = PLC "HMI_Interface.Data".meta AT %DB1.DBW0, 100 ms

Template "Navigation" 800x480
   ScreenModuleView "Navigation_1" at 0,0 size 800x65; ScreenModuleType ""
      Guid_{11997190-7796} <- "HMI_Interface.Data_navigation"
      on Guid_{11997190-7994}: ActivateScreen("02_Materials", 0)
      on Guid_{11997190-7997}: ActivateScreen("01_Wires", 0)

screen "01_Wires" 800x480, template "Navigation"
   on GenerateScreen: SetTag("screen_number", 1)
   ScreenModuleView "heat" at 100,75 size 600x65; Guid_{11997190-6447} 'HEAT'; ScreenModuleType ""
      Guid_{11997190-5401} <- "heat"
   ScreenModuleView "label" at 100,140 size 600x65; Guid_{11997190-7215} 'FEET'; ScreenModuleType ""
      Guid_{11997190-5401} <- "header"
   ScreenModuleView "divider" at 100,205 size 600x5; ScreenModuleType ""
      Guid_{11997190-7534} <- "divider"
   ScreenModuleView "carbon" at 100,210 size 600x65; Guid_{11997190-6447} 'CARBON'; ScreenModuleType ""
      Guid_{11997190-5401} <- "carbon"
   ScreenModuleView "calcium_silicon" at 100,275 size 600x65; Guid_{11997190-6447} 'CAL/SIL'; ScreenModuleType ""
      Guid_{11997190-5401} <- "calcium_silicon"
   ScreenModuleView "aluminium" at 100,340 size 600x65; Guid_{11997190-6447} 'ALUMINIUM'; ScreenModuleType ""
      Guid_{11997190-5401} <- "aluminum"
   ScreenModuleView "sulfur" at 100,405 size 600x65; Guid_{11997190-6447} 'SULFUR'; ScreenModuleType ""
      Guid_{11997190-5401} <- "sulfur"
   ScreenModuleView "bottom_border" at 100,470 size 600x5; ScreenModuleType ""
      Guid_{11997190-7534} <- "bottom_border"
   Rectangle "Rectangle_1" at 0,65 size 800x415
      Appearance <- "color"
      Visibility <- "visible"

screen "02_Materials" 800x480, template "Navigation"
   on GenerateScreen: SetTag("screen_number", 2)
   ScreenModuleView "heat" at 100,87 size 600x40; Guid_{11997190-6447} 'HEAT'; ScreenModuleType ""
      Guid_{11997190-5401} <- "heat"
   ScreenModuleView "material_label" at 100,127 size 600x40; ScreenModuleType ""
      Guid_{11997190-5401} <- "header"
   ScreenModuleView "divider" at 100,167 size 600x5; ScreenModuleType ""
      Guid_{11997190-7534} <- "divider"
   ScreenModuleView "manganese" at 100,172 size 600x40; Guid_{11997190-6447} 'MANGANESE'; ScreenModuleType ""
      Guid_{11997190-5401} <- "manganese"
   ScreenModuleView "silicon" at 100,212 size 600x40; Guid_{11997190-6447} 'SILICON'; ScreenModuleType ""
      Guid_{11997190-5401} <- "silicon"
   ScreenModuleView "chromium" at 100,252 size 600x40; Guid_{11997190-6447} 'CHROMIUM'; ScreenModuleType ""
      Guid_{11997190-5401} <- "chromium"
   ScreenModuleView "vanadium" at 100,292 size 600x40; Guid_{11997190-6447} 'VANADIUM'; ScreenModuleType ""
      Guid_{11997190-5401} <- "vanadium"
   ScreenModuleView "nickel" at 100,332 size 600x40; Guid_{11997190-6447} 'NICKEL'; ScreenModuleType ""
      Guid_{11997190-5401} <- "nickel"
   ScreenModuleView "molybdenum" at 100,372 size 600x40; Guid_{11997190-6447} 'MOLYBDENUM'; ScreenModuleType ""
      Guid_{11997190-5401} <- "molybdenum"
   ScreenModuleView "bottom_border" at 100,452 size 600x5; ScreenModuleType ""
      Guid_{11997190-7534} <- "bottom_border"
   ScreenModuleView "custom" at 100,412 size 600x40; ScreenModuleType ""
      Guid_{11997190-5401} <- "custom"
   Rectangle "screen_background" at 0,65 size 800x415
      Appearance <- "color"
      Visibility <- "visible"
*)

(* ===== HMI "HMI_RT_1" =====
system functions are stored by id; their names below are inferred from use

ScreenModuleEditorView "Row_Wire" 400x50
   Rectangle "Border" at 0,0 size 400x50
      Appearance <- "interface.background_animate"
   IOField "IOF R0 C0" at 5,5 size 190x45; FormatPattern ????????????????????
      ProcessValue <- "text_label"
      Appearance <- "interface.cell_0_animate"
      ObjectEnable <- "interface.cell_0_enable"
      Visibility <- "interface.cell_0_visible"
   IOField "IOF R0 C1" at 200,5 size 195x45; FormatPattern 9999999
      on OnFinishInput: SetBit("interface.cell_1_input_finished")
      Visibility <- "interface.cell_1_visible"
      ObjectEnable <- "interface.cell_1_enable"
      Appearance <- "interface.cell_1_animate"
*)

(* ===== HMI "HMI_RT_1" =====
system functions are stored by id; their names below are inferred from use

ScreenModuleEditorView "Row_Wire" 400x50
   Rectangle "Border" at 0,0 size 400x50
      Appearance <- "interface.background_animate"
      Visibility <- "interface.background_visible"
   IOField "IOF R0 C0" at 5,5 size 190x45; FormatPattern ????????????????????
      Appearance <- "interface.cell_0_animate"
      ProcessValue <- "text_label"
      Visibility <- "interface.cell_0_visible"
      ObjectEnable <- "interface.cell_0_enable"
   IOField "IOF R0 C1" at 200,5 size 195x45; FormatPattern 9999999
      on OnFinishInput: SetBit("interface.cell_1_input_finished")
      Visibility <- "interface.cell_1_visible"
      Appearance <- "interface.cell_1_animate"
      ObjectEnable <- "interface.cell_1_enable"
*)

(* ===== HMI "HMI_RT_1" =====
system functions are stored by id; their names below are inferred from use

ScreenModuleEditorView "Row_Wire" 400x50
   Rectangle "Border" at 0,0 size 400x50
      Visibility <- "interface.background_visible"
      Appearance <- "interface.background_animate"
   IOField "IOF R0 C0" at 5,5 size 190x45; FormatPattern ????????????????????
      Appearance <- "interface.cell_0_animate"
      Visibility <- "interface.cell_0_visible"
      ObjectEnable <- "interface.cell_0_enable"
      ProcessValue <- "interface.cell_0_value"
   IOField "IOF R0 C1" at 200,5 size 195x45; FormatPattern 9999999
      on OnFinishInput: SetBit("interface.cell_1_input_finished")
      Visibility <- "interface.cell_1_visible"
      Appearance <- "interface.cell_1_animate"
      ObjectEnable <- "interface.cell_1_enable"
*)

(* ===== HMI "HMI_RT_1" =====
system functions are stored by id; their names below are inferred from use

ScreenModuleEditorView "Row_Wire" 400x50
   Rectangle "Border" at 0,0 size 400x50
      Visibility <- "interface.background_visible"
      Appearance <- "interface.background_animate"
   IOField "IOF R0 C0" at 5,5 size 190x45; FormatPattern ????????????????????
      Appearance <- "interface.cell_0_animate"
      Visibility <- "interface.cell_0_visible"
      ProcessValue <- "interface.cell_0_value"
      ObjectEnable <- "interface.cell_0_enable"
   IOField "IOF R0 C1" at 200,5 size 195x45; FormatPattern 9999999
      on OnFinishInput: SetBit("interface.cell_1_input_finished")
      Visibility <- "interface.cell_1_visible"
      Appearance <- "interface.cell_1_animate"
      ObjectEnable <- "interface.cell_1_enable"
*)

(* ===== HMI "HMI_RT_1" =====
system functions are stored by id; their names below are inferred from use

ScreenModuleEditorView "Row_Wire" 400x65
   Rectangle "Border" at 0,0 size 400x65
      Visibility <- "interface.background_visible"
      Appearance <- "interface.background_animate"
   TextField "TF R0 C0" at 5,5 size 190x60; Text 'Text'
      Visibility <- "interface.cell_0_visible"
   IOField "IOF R0 C1" at 200,5 size 195x60; FormatPattern 9999999
      on OnFinishInput: SetBit("interface.cell_1_input_finished")
      Visibility <- "interface.cell_1_visible"
      ObjectEnable <- "interface.cell_1_enable"
*)

(* ===== HMI "HMI_RT_1" =====
system functions are stored by id; their names below are inferred from use

ScreenModuleEditorView "Row_Wire" 600x65
   Rectangle "Border" at 0,0 size 600x65
      Visibility <- "interface.background_visible"
      Appearance <- "interface.background_animate"
   TextField "TF R0 C0" at 5,5 size 360x60; Text 'CARBON WIRE'
      Visibility <- "interface.cell_0_visible"
   IOField "IOF R0 C1" at 370,5 size 225x60; FormatPattern 9999999
      on OnFinishInput: SetBit("interface.cell_1_input_finished")
      Visibility <- "interface.cell_1_visible"
      ObjectEnable <- "interface.cell_1_enable"
*)

(* ===== HMI "HMI_RT_1" =====
system functions are stored by id; their names below are inferred from use

ScreenModuleEditorView "Row_Wire" 600x65
   Rectangle "Border" at 0,0 size 600x65
      Visibility <- "interface.background_visible"
      Appearance <- "interface.background_animate"
   TextField "TF R0 C0" at 5,5 size 360x60; Text 'CARBON WIRE'
      Visibility <- "interface.cell_0_visible"
      Appearance <- "interface.cell_0_animate"
   IOField "IOF R0 C1" at 370,5 size 225x60; FormatPattern 9999999
      on OnFinishInput: SetBit("interface.cell_1_input_finished")
      Visibility <- "interface.cell_1_visible"
      ObjectEnable <- "interface.cell_1_enable"
      Appearance <- "interface.cell_1_animate"
*)

(* ===== HMI "HMI_RT_1" =====
system functions are stored by id; their names below are inferred from use

ScreenModuleEditorView "Row_Wire_Label" 600x65
   Rectangle "Border" at 0,0 size 600x65
      Visibility <- "interface.background_visible"
      Appearance <- "interface.background_animate"
   TextField "TF R0 C0" at 5,5 size 360x60; Text 'CARBON WIRE'
      Visibility <- "interface.cell_0_visible"
      Appearance <- "interface.cell_0_animate"
   IOField "IOF R0 C1" at 370,5 size 225x60; FormatPattern 9999999
      on OnFinishInput: SetBit("interface.cell_1_input_finished")
      Visibility <- "interface.cell_1_visible"
      Appearance <- "interface.cell_1_animate"
      ObjectEnable <- "interface.cell_1_enable"
*)

(* ===== HMI "HMI_RT_1" =====

ScreenModuleEditorView "Row_Wire_Label" 600x65
   Rectangle "Border" at 0,0 size 600x65
      Visibility <- "interface.background_visible"
      Appearance <- "interface.background_animate"
   TextField "TF R0 C0" at 5,5 size 360x60; Text 'WIRE'
      Visibility <- "interface.cell_0_visible"
      Appearance <- "interface.cell_0_animate"
   TextField "TF R0 C1" at 370,5 size 225x60; Text 'LENGTH'
      Visibility <- "interface.cell_1_visible"
      Appearance <- "interface.cell_1_animate"
*)

(* ===== HMI "HMI_RT_1" =====

ScreenModuleEditorView "Divider" 600x5
   Line "line" at 10,2 size 580x0
      Appearance <- "interface.line_animate"
      Visibility <- "interface.line_visible"
   Rectangle "background" at 0,0 size 600x5
      Appearance <- "interface.background_animate"
      Visibility <- "interface.background_visible"
*)

(* ===== HMI "HMI_RT_1" =====
system functions are stored by id; their names below are inferred from use

ScreenModuleEditorView "Navigation" 800x65
   Button "Wire" at 5,5 size 390x60; TextOff 'WIRE'
      Appearance <- "interface.wire_animate"
      on Press: function_b14e0dd5("interface.wire_actuate", 0)
   Button "Material" at 400,5 size 390x60; TextOff 'MATERIAL'
      Appearance <- "interface.material_animate"
      on Press: function_b14e0dd5("interface.material_actuate", 0)
   Rectangle "Wire_Cover" at 10,60 size 380x5
      Visibility <- "interface.wire_cover_visible"
   Rectangle "Material_Cover" at 405,60 size 380x5
      Visibility <- "interface.material_cover_visible"
*)

(* ===== HMI "HMI_RT_1" =====
system functions are stored by id; their names below are inferred from use

ScreenModuleEditorView "Navigation" 800x65
   Button "Wire" at 5,5 size 390x60; TextOff 'WIRE'
      on Press: function_b14e0dd5("interface.wire_actuate", 0)
      Appearance <- "interface.wire_animate"
   Button "Material" at 400,5 size 390x60; TextOff 'MATERIAL'
      on Press: function_b14e0dd5("interface.material_actuate", 0)
      Appearance <- "interface.material_animate"
   Rectangle "Wire_Cover" at 10,60 size 380x5
      Visibility <- "interface.wire_cover_visible"
   Rectangle "Material_Cover" at 405,60 size 380x5
      Visibility <- "interface.material_cover_visible"
*)

(* ===== HMI "HMI_RT_1" =====
system functions are stored by id; their names below are inferred from use

ScreenModuleEditorView "Navigation" 800x65
   Button "Wire" at 5,5 size 392x60; TextOff 'WIRE'
      on Press: function_b14e0dd5("interface.wire_actuate", 0)
      Appearance <- "interface.wire_animate"
   Button "Material" at 402,5 size 393x60; TextOff 'MATERIAL'
      on Press: function_b14e0dd5("interface.material_actuate", 0)
      Appearance <- "interface.material_animate"
   Rectangle "Wire_Cover" at 10,60 size 382x5
      Visibility <- "interface.wire_cover_visible"
   Rectangle "Material_Cover" at 407,60 size 383x5
      Visibility <- "interface.material_cover_visible"
*)

(* ===== HMI "HMI_RT_1" =====
system functions are stored by id; their names below are inferred from use

ScreenModuleEditorView "Row_Material" 600x65
   Rectangle "Border" at 0,0 size 600x65
      Visibility <- "interface.background_visible"
      Appearance <- "interface.background_animate"
   TextField "TF R0 C0" at 5,5 size 360x60; Text 'CARBON WIRE'
      Visibility <- "interface.cell_0_visible"
      Appearance <- "interface.cell_0_animate"
   IOField "IOF R0 C1" at 370,5 size 225x60; FormatPattern 9999999
      on OnFinishInput: SetBit("interface.cell_1_input_finished")
      Visibility <- "interface.cell_1_visible"
      Appearance <- "interface.cell_1_animate"
      ObjectEnable <- "interface.cell_1_enable"
*)

(* ===== HMI "HMI_RT_1" =====
system functions are stored by id; their names below are inferred from use

ScreenModuleEditorView "Row_Material" 600x40
   Rectangle "Border" at 0,0 size 600x40
      Visibility <- "interface.background_visible"
      Appearance <- "interface.background_animate"
   IOField "IOF R0 C1" at 370,5 size 225x35; FormatPattern 9999999
      on OnFinishInput: SetBit("interface.cell_1_input_finished")
      Visibility <- "interface.cell_1_visible"
      Appearance <- "interface.cell_1_animate"
      ObjectEnable <- "interface.cell_1_enable"
   TextField "TF R0 C0" at 5,5 size 360x35; Text 'MOLYBDENUM'
      Visibility <- "interface.cell_0_visible"
      Appearance <- "interface.cell_0_animate"
*)

(* ===== HMI "HMI_RT_1" =====
system functions are stored by id; their names below are inferred from use

ScreenModuleEditorView "Row_Custom" 600x40
   Rectangle "Border" at 0,0 size 600x40
      Visibility <- "interface.background_visible"
      Appearance <- "interface.background_animate"
   IOField "IOF R0 C1" at 370,5 size 225x35; FormatPattern 9999999
      on OnFinishInput: SetBit("interface.cell_1_input_finished")
      Visibility <- "interface.cell_1_visible"
      Appearance <- "interface.cell_1_animate"
      ObjectEnable <- "interface.cell_1_enable"
   TextField "TF R0 C0" at 5,5 size 360x35; Text 'MOLYBDENUM'
      Visibility <- "interface.cell_0_visible"
      Appearance <- "interface.cell_0_animate"
*)

(* ===== HMI "HMI_RT_1" =====
system functions are stored by id; their names below are inferred from use

ScreenModuleEditorView "Row_Custom" 600x40
   Rectangle "Border" at 0,0 size 600x40
      Visibility <- "interface.background_visible"
      Appearance <- "interface.background_animate"
   IOField "IOF R0 C0" at 5,5 size 360x35; FormatPattern ???????????????
      on OnFinishInput: SetBit("interface.cell_0_input_finished")
      Appearance <- "interface.cell_0_animate"
      ObjectEnable <- "interface.cell_0_enable"
      Visibility <- "interface.cell_0_visible"
   IOField "IOF R0 C1" at 370,5 size 225x35; FormatPattern 9999999
      on OnFinishInput: SetBit("interface.cell_1_input_finished")
      Visibility <- "interface.cell_1_visible"
      Appearance <- "interface.cell_1_animate"
      ObjectEnable <- "interface.cell_1_enable"
*)

(* ===== HMI "HMI_RT_1" =====
system functions are stored by id; their names below are inferred from use

ScreenModuleEditorView "Row_Material_Label" 600x40
   Rectangle "Border" at 0,0 size 600x40
      Visibility <- "interface.background_visible"
      Appearance <- "interface.background_animate"
   IOField "IOF R0 C1" at 370,5 size 225x35; FormatPattern 9999999
      on OnFinishInput: SetBit("interface.cell_1_input_finished")
      Visibility <- "interface.cell_1_visible"
      Appearance <- "interface.cell_1_animate"
      ObjectEnable <- "interface.cell_1_enable"
   TextField "TF R0 C0" at 5,5 size 360x35; Text 'MOLYBDENUM'
      Visibility <- "interface.cell_0_visible"
      Appearance <- "interface.cell_0_animate"
*)

(* ===== HMI "HMI_RT_1" =====

ScreenModuleEditorView "Row_Material_Label" 600x40
   Rectangle "Border" at 0,0 size 600x40
      Visibility <- "interface.background_visible"
      Appearance <- "interface.background_animate"
   TextField "TF R0 C0" at 5,5 size 360x35; Text 'MATERIAL'
      Visibility <- "interface.cell_0_visible"
      Appearance <- "interface.cell_0_animate"
   TextField "TF R0 C1" at 370,5 size 225x35; Text 'BAGS'
      Appearance <- "interface.cell_1_animate"
      Visibility <- "interface.cell_1_visible"
*)

(* ===== HMI "HMI_RT_1" =====
system functions are stored by id; their names below are inferred from use

ScreenModuleEditorView "Row_Wire" 600x65
   Rectangle "Border" at 0,0 size 600x65
      Visibility <- "interface.background_visible"
   TextField "TF R0 C0" at 5,5 size 360x60; Text 'CARBON WIRE'
      Visibility <- "interface.cell_0_visible"
   IOField "IOF R0 C1" at 370,5 size 225x60; FormatPattern 9999999
      on OnFinishInput: SetBit("interface.cell_1_input_finished")
      Visibility <- "interface.cell_1_visible"
      Appearance <- "interface.cell_1_animate"
      ObjectEnable <- "interface.cell_1_enable"
      on Activate: SetBit("interface.cell_1_active")
      on Deactivate: ResetBit("interface.cell_1_active")
*)

(* ===== HMI "HMI_RT_1" =====

ScreenModuleEditorView "Divider" 600x5
   Line "line" at 10,2 size 580x0
      Visibility <- "interface.line_visible"
      Appearance <- "interface.line_animate"
   Rectangle "background" at 0,0 size 600x5
      Visibility <- "interface.background_visible"
      Appearance <- "interface.background_animate"
*)

(* ===== HMI "HMI_RT_1" =====
system functions are stored by id; their names below are inferred from use

ScreenModuleEditorView "Row_Material" 600x40
   Rectangle "Border" at 0,0 size 600x40
      Visibility <- "interface.background_visible"
      Appearance <- "interface.background_animate"
   IOField "IOF R0 C1" at 370,5 size 225x35; FormatPattern 9999999
      on OnFinishInput: SetBit("interface.cell_1_input_finished")
      Visibility <- "interface.cell_1_visible"
      Appearance <- "interface.cell_1_animate"
      ObjectEnable <- "interface.cell_1_enable"
   TextField "TF R0 C0" at 5,5 size 360x35; Text 'MOLYBDENUM'
      Visibility <- "interface.cell_0_visible"
      Appearance <- "interface.cell_0_animate"
*)

(* ===== HMI "HMI_RT_1" =====
system functions are stored by id; their names below are inferred from use

ScreenModuleEditorView "Navigation" 800x65
   Button "Wire" at 5,5 size 392x60; TextOff 'WIRE'
      on Press: function_b14e0dd5("interface.wire_actuate", 0)
      Appearance <- "interface.wire_animate"
      ObjectEnable <- "interface.wire_enable"
      Visibility <- "interface.wire_visible"
   Button "Material" at 402,5 size 393x60; TextOff 'MATERIAL'
      on Press: function_b14e0dd5("interface.material_actuate", 0)
      Appearance <- "interface.material_animate"
      ObjectEnable <- "interface.material_enable"
      Visibility <- "interface.material_visible"
   Rectangle "Background" at 0,0 size 800x65
      Appearance <- "interface.background_animate"
      Visibility <- "interface.background_visible"
   Rectangle "Wire_Cover" at 10,60 size 382x5
      Visibility <- "interface.wire_cover_visible"
      Appearance <- "interface.wire_cover_animate"
   Rectangle "Material_Cover" at 407,60 size 383x5
      Visibility <- "interface.material_cover_visible"
      Appearance <- "interface.material_cover_animate"
   Line "Bottom_Line" at 0,62 size 800x0
      Appearance <- "interface.bottom_line_animate"
      Visibility <- "interface.bottom_line_visible"
*)

(* ===== HMI "HMI_RT_1" =====
system functions are stored by id; their names below are inferred from use

ScreenModuleEditorView "Navigation" 800x65
   Button "Wire" at 5,5 size 392x60; TextOff 'WIRE'
      on Press: function_b14e0dd5("interface.wire_actuate", 0)
      Appearance <- "interface.wire_animate"
      ObjectEnable <- "interface.wire_enable"
      Visibility <- "interface.wire_visible"
   Button "Material" at 402,5 size 393x60; TextOff 'MATERIAL'
      on Press: function_b14e0dd5("interface.material_actuate", 0)
      Appearance <- "interface.material_animate"
      ObjectEnable <- "interface.material_enable"
      Visibility <- "interface.material_visible"
   Rectangle "Background" at 0,0 size 800x65
      Visibility <- "interface.background_visible"
      Appearance <- "interface.background_animate"
   Rectangle "Wire_Cover" at 10,60 size 382x5
      Visibility <- "interface.wire_cover_visible"
      Appearance <- "interface.wire_cover_animate"
   Rectangle "Material_Cover" at 407,60 size 383x5
      Visibility <- "interface.material_cover_visible"
      Appearance <- "interface.material_cover_animate"
   Line "Bottom_Line" at 0,62 size 800x0
      Visibility <- "interface.bottom_line_visible"
      Appearance <- "interface.bottom_line_animate"
*)

(* ===== HMI "HMI_RT_1" =====
system functions are stored by id; their names below are inferred from use

ScreenModuleEditorView "Navigation" 800x65
   Button "Wire" at 5,5 size 392x60; TextOff 'WIRE'
      on Press: function_b14e0dd5("interface.wire_actuate", 0)
      Appearance <- "interface.wire_animate"
      ObjectEnable <- "interface.wire_enable"
      Visibility <- "interface.wire_visible"
   Button "Material" at 402,5 size 393x60; TextOff 'MATERIAL'
      on Press: function_b14e0dd5("interface.material_actuate", 0)
      Appearance <- "interface.material_animate"
      ObjectEnable <- "interface.material_enable"
      Visibility <- "interface.material_visible"
   Rectangle "Background" at 0,0 size 800x65
      Visibility <- "interface.background_visible"
      Appearance <- "interface.background_animate"
   Rectangle "Wire_Cover" at 10,60 size 382x5
      Visibility <- "interface.wire_cover_visible"
      Appearance <- "interface.wire_cover_animate"
   Rectangle "Material_Cover" at 407,60 size 383x5
      Visibility <- "interface.material_cover_visible"
      Appearance <- "interface.material_cover_animate"
   Line "Bottom_Line" at 0,62 size 800x0
      Visibility <- "interface.bottom_line_visible"
      Appearance <- "interface.bottom_line_animate"
*)

(* ===== HMI "HMI_RT_1" =====
system functions are stored by id; their names below are inferred from use

ScreenModuleEditorView "Navigation" 800x65
   Button "Wire" at 5,5 size 392x60; TextOff 'WIRE'
      on Press: function_b14e0dd5("interface.wire_actuate", 0)
      Appearance <- "interface.wire_animate"
      ObjectEnable <- "interface.wire_enable"
      Visibility <- "interface.wire_visible"
   Button "Material" at 402,5 size 393x60; TextOff 'MATERIAL'
      on Press: function_b14e0dd5("interface.material_actuate", 0)
      Appearance <- "interface.material_animate"
      ObjectEnable <- "interface.material_enable"
      Visibility <- "interface.material_visible"
   Rectangle "Background" at 0,0 size 800x65
      Visibility <- "interface.background_visible"
      Appearance <- "interface.background_animate"
   Rectangle "Wire_Cover" at 10,60 size 382x5
      Visibility <- "interface.wire_cover_visible"
      Appearance <- "interface.wire_cover_animate"
   Rectangle "Material_Cover" at 407,60 size 383x5
      Visibility <- "interface.material_cover_visible"
      Appearance <- "interface.material_cover_animate"
   Line "Bottom_Line" at 0,62 size 800x0
      Visibility <- "interface.bottom_line_visible"
      Appearance <- "interface.bottom_line_animate"
*)

(* ===== HMI "HMI_RT_1" =====
system functions are stored by id; their names below are inferred from use

ScreenModuleEditorView "Navigation" 800x65
   Button "Wire" at 5,5 size 392x60; TextOff 'WIRE'
      on Press: function_b14e0dd5("interface.wire_actuate", 0)
      Appearance <- "interface.wire_animate"
      ObjectEnable <- "interface.wire_enable"
      Visibility <- "interface.wire_visible"
   Button "Material" at 402,5 size 393x60; TextOff 'MATERIAL'
      on Press: function_b14e0dd5("interface.material_actuate", 0)
      Appearance <- "interface.material_animate"
      ObjectEnable <- "interface.material_enable"
      Visibility <- "interface.material_visible"
   Rectangle "Background" at 0,0 size 800x65
      Visibility <- "interface.background_visible"
      Appearance <- "interface.background_animate"
   Rectangle "Wire_Cover" at 10,60 size 382x5
      Visibility <- "interface.wire_cover_visible"
      Appearance <- "interface.wire_cover_animate"
   Rectangle "Material_Cover" at 407,60 size 383x5
      Visibility <- "interface.material_cover_visible"
      Appearance <- "interface.material_cover_animate"
   Line "Bottom_Line" at 0,62 size 800x0
      Visibility <- "interface.bottom_line_visible"
      Appearance <- "interface.bottom_line_animate"
*)

(* ===== HMI "HMI_RT_1" =====

ScreenModuleEditorView "Row_Wire_Label" 600x65
   Rectangle "Border" at 0,0 size 600x65
      Visibility <- "interface.background_visible"
      Appearance <- "interface.background_animate"
   TextField "TF R0 C0" at 5,5 size 360x60; Text 'WIRE'
      Visibility <- "interface.cell_0_visible"
      Appearance <- "interface.cell_0_animate"
   TextField "TF R0 C1" at 370,5 size 225x60; Text 'LENGTH'
      Visibility <- "interface.cell_1_visible"
      Appearance <- "interface.cell_1_animate"
*)

(* ===== HMI "HMI_RT_1" =====
system functions are stored by id; their names below are inferred from use

ScreenModuleEditorView "Row_Wire" 600x65
   Rectangle "Border" at 0,0 size 600x65
      Visibility <- "interface.background_visible"
      Appearance <- "interface.background_animate"
   TextField "TF R0 C0" at 5,5 size 360x60; Text 'CARBON WIRE'
      Visibility <- "interface.cell_0_visible"
      Appearance <- "interface.cell_0_animate"
   IOField "IOF R0 C1" at 370,5 size 225x60; FormatPattern 9999999
      on OnFinishInput: SetBit("interface.cell_1_input_finished")
      on Deactivate: ResetBit("interface.cell_1_active")
      on Activate: SetBit("interface.cell_1_active")
      Visibility <- "interface.cell_1_visible"
      ObjectEnable <- "interface.cell_1_enable"
      Appearance <- "interface.cell_1_animate"
*)

(* ===== HMI "HMI_RT_1" =====

ScreenModuleEditorView "Row_Wire_Label" 600x65
   Rectangle "Border" at 0,0 size 600x65
      Visibility <- "interface.background_visible"
      Appearance <- "interface.background_animate"
   TextField "TF R0 C0" at 5,5 size 360x60; Text 'WIRE'
      Visibility <- "interface.cell_0_visible"
      Appearance <- "interface.cell_0_animate"
   TextField "TF R0 C1" at 370,5 size 225x60; Text 'LENGTH'
      Visibility <- "interface.cell_1_visible"
      Appearance <- "interface.cell_1_animate"
*)

(* ===== HMI "HMI_RT_1" =====
system functions are stored by id; their names below are inferred from use

